// TIA Portal V17 export
// export: Created 2025-04-25T10:07:11.7056769Z, ExportSetting WithDefaults, DisplayName Totally Integrated Automation Portal, DisplayVersion V17 Update 8, DisplayName TIA Portal Openness, DisplayVersion V17 Update 8, DisplayName TIA Portal Version Control Interface, DisplayVersion V17, DisplayName SINAMICS Startdrive Advanced, DisplayVersion V17 SP2, DisplayName SINAMICS Startdrive G110M, G120, G120C, G120D, G120P, G115D, DisplayVersion V17 SP2, DisplayName SINAMICS Startdrive G130, G150, S120, S150, SINAMICS MV, S210, DisplayVersion V17 SP2, DisplayName STEP 7 Professional, DisplayVersion V17 Update 8, DisplayName SINUMERIK ONE STEP 7 Toolbox, DisplayVersion V17 Update 12, DisplayName SINUMERIK 840D sl STEP 7 Toolbox, DisplayVersion V17 Update 12, DisplayName STEP 7 Safety, DisplayVersion V17 Update 6, DisplayName WinCC Advanced / Unified PC, DisplayVersion V17 Update 8
FUNCTION "FC353_NCK_M_CH3_UNIT_1_STA_4" : Void   // FC353, LAD
TITLE = Channel 1 data
{ S7_Optimized_Access := 'FALSE' }
AUTHOR : ETXETAR
VERSION : 1.0
// stored: AutoNumber false, IsIECCheckEnabled false, SetENOAutomatically false, UDAEnableTagReadback false
   VAR_TEMP
      auxm3 : Bool;
      auxm5 : Bool;
   END_VAR
   VAR_TEMP   // added for the SCL form of the ladder/FBD networks
      _w1 : Bool;
      _w2 : Bool;
   END_VAR
BEGIN

REGION Network 1: CALL FB331 M CODE EXTENDED CH4 / M CODE EXTENDED CHANNEL 2
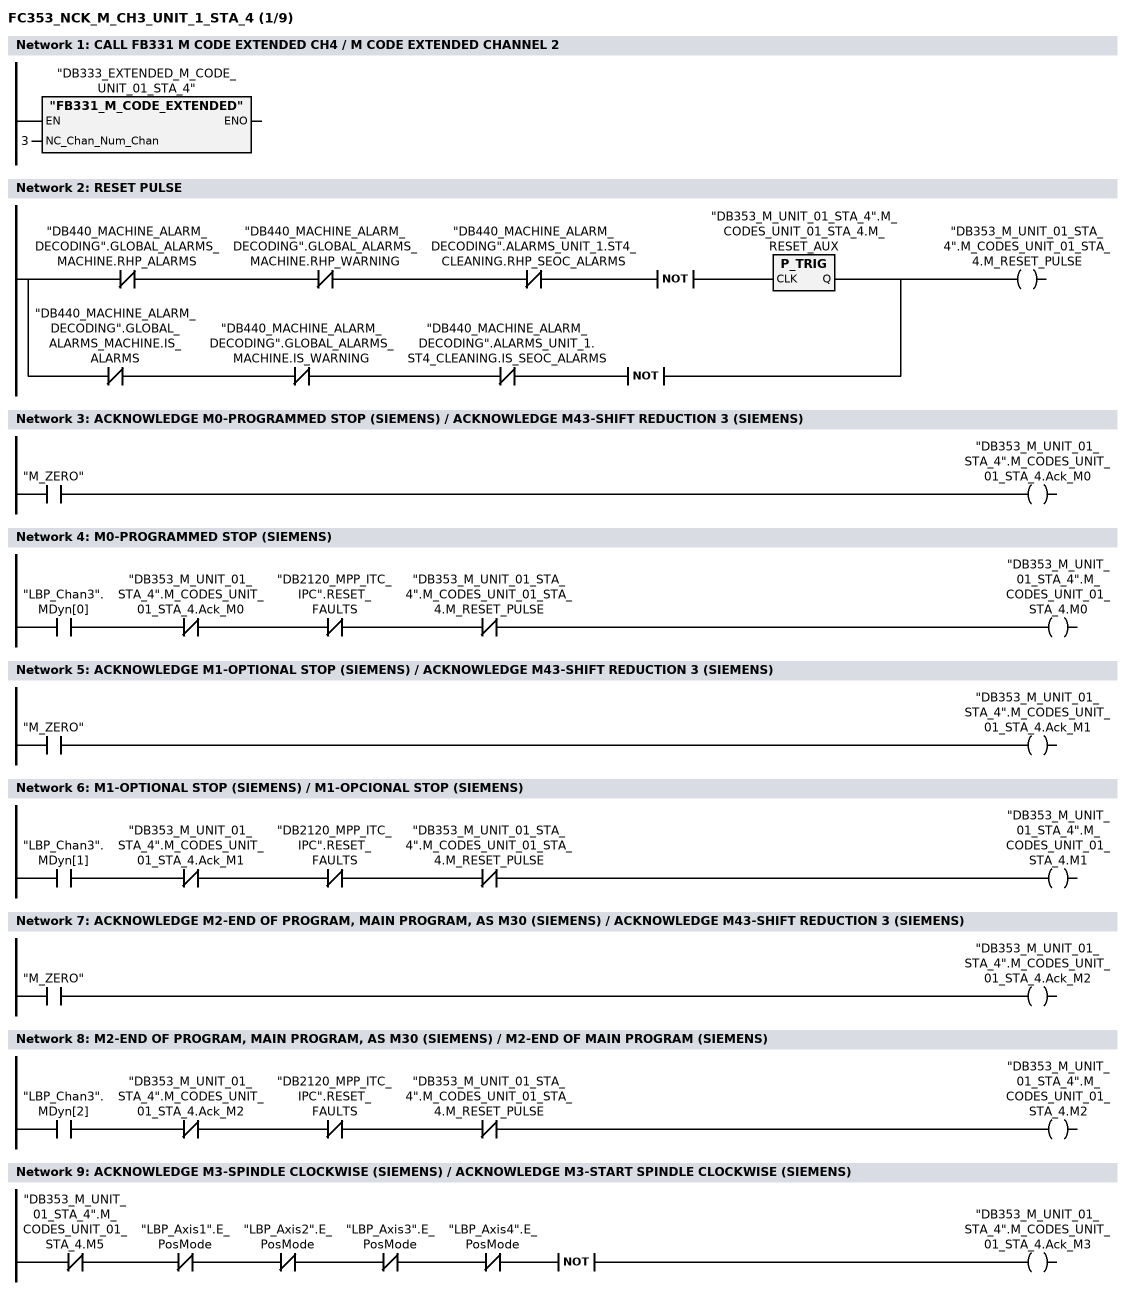
   RUNG wire#powerrail
      "DB333_EXTENDED_M_CODE_UNIT_01_STA_4"(NC_Chan_Num_Chan := 3)
   END_RUNG
   // the same network as SCL:
   "DB333_EXTENDED_M_CODE_UNIT_01_STA_4"(NC_Chan_Num_Chan := 3);   // "FB331_M_CODE_EXTENDED"
END_REGION

REGION Network 2: RESET PULSE
   RUNG wire#powerrail
      I_Contact( "DB440_MACHINE_ALARM_DECODING".GLOBAL_ALARMS_MACHINE.RHP_ALARMS )
      I_Contact( "DB440_MACHINE_ALARM_DECODING".GLOBAL_ALARMS_MACHINE.RHP_WARNING )
      I_Contact( "DB440_MACHINE_ALARM_DECODING".ALARMS_UNIT_1.ST4_CLEANING.RHP_SEOC_ALARMS )
      Not()
      P_Trig( "DB353_M_UNIT_01_STA_4".M_CODES_UNIT_01_STA_4.M_RESET_AUX )
      wire#w1
      Coil( "DB353_M_UNIT_01_STA_4".M_CODES_UNIT_01_STA_4.M_RESET_PULSE )
   END_RUNG
   RUNG wire#powerrail
      I_Contact( "DB440_MACHINE_ALARM_DECODING".GLOBAL_ALARMS_MACHINE.IS_ALARMS )
      I_Contact( "DB440_MACHINE_ALARM_DECODING".GLOBAL_ALARMS_MACHINE.IS_WARNING )
      I_Contact( "DB440_MACHINE_ALARM_DECODING".ALARMS_UNIT_1.ST4_CLEANING.IS_SEOC_ALARMS )
      Not()
   END_RUNG wire#w1
   // the same network as SCL:
   #_w1 := NOT (NOT "DB440_MACHINE_ALARM_DECODING".GLOBAL_ALARMS_MACHINE.RHP_ALARMS AND NOT "DB440_MACHINE_ALARM_DECODING".GLOBAL_ALARMS_MACHINE.RHP_WARNING AND NOT "DB440_MACHINE_ALARM_DECODING".ALARMS_UNIT_1.ST4_CLEANING.RHP_SEOC_ALARMS);
   #_w2 := #_w1 AND NOT "DB353_M_UNIT_01_STA_4".M_CODES_UNIT_01_STA_4.M_RESET_AUX;   // rising edge
   "DB353_M_UNIT_01_STA_4".M_CODES_UNIT_01_STA_4.M_RESET_AUX := #_w1;
   "DB353_M_UNIT_01_STA_4".M_CODES_UNIT_01_STA_4.M_RESET_PULSE := #_w2 OR NOT (NOT "DB440_MACHINE_ALARM_DECODING".GLOBAL_ALARMS_MACHINE.IS_ALARMS AND NOT "DB440_MACHINE_ALARM_DECODING".GLOBAL_ALARMS_MACHINE.IS_WARNING AND NOT "DB440_MACHINE_ALARM_DECODING".ALARMS_UNIT_1.ST4_CLEANING.IS_SEOC_ALARMS);
END_REGION

REGION Network 3: ACKNOWLEDGE M0-PROGRAMMED STOP (SIEMENS) / ACKNOWLEDGE M43-SHIFT REDUCTION 3 (SIEMENS)
   RUNG wire#powerrail
      Contact( "M_ZERO" )
      Coil( "DB353_M_UNIT_01_STA_4".M_CODES_UNIT_01_STA_4.Ack_M0 )
   END_RUNG
   // the same network as SCL:
   "DB353_M_UNIT_01_STA_4".M_CODES_UNIT_01_STA_4.Ack_M0 := "M_ZERO";
END_REGION

REGION Network 4: M0-PROGRAMMED STOP (SIEMENS)
   RUNG wire#powerrail
      Contact( "LBP_Chan3".MDyn[0] )
      I_Contact( "DB353_M_UNIT_01_STA_4".M_CODES_UNIT_01_STA_4.Ack_M0 )
      I_Contact( "DB2120_MPP_ITC_IPC".RESET_FAULTS )
      I_Contact( "DB353_M_UNIT_01_STA_4".M_CODES_UNIT_01_STA_4.M_RESET_PULSE )
      Coil( "DB353_M_UNIT_01_STA_4".M_CODES_UNIT_01_STA_4.M0 )
   END_RUNG
   // the same network as SCL:
   "DB353_M_UNIT_01_STA_4".M_CODES_UNIT_01_STA_4.M0 := "LBP_Chan3".MDyn[0] AND NOT "DB353_M_UNIT_01_STA_4".M_CODES_UNIT_01_STA_4.Ack_M0 AND NOT "DB2120_MPP_ITC_IPC".RESET_FAULTS AND NOT "DB353_M_UNIT_01_STA_4".M_CODES_UNIT_01_STA_4.M_RESET_PULSE;
END_REGION

REGION Network 5: ACKNOWLEDGE M1-OPTIONAL STOP (SIEMENS) / ACKNOWLEDGE M43-SHIFT REDUCTION 3 (SIEMENS)
   RUNG wire#powerrail
      Contact( "M_ZERO" )
      Coil( "DB353_M_UNIT_01_STA_4".M_CODES_UNIT_01_STA_4.Ack_M1 )
   END_RUNG
   // the same network as SCL:
   "DB353_M_UNIT_01_STA_4".M_CODES_UNIT_01_STA_4.Ack_M1 := "M_ZERO";
END_REGION

REGION Network 6: M1-OPTIONAL STOP (SIEMENS) / M1-OPCIONAL STOP (SIEMENS)
   RUNG wire#powerrail
      Contact( "LBP_Chan3".MDyn[1] )
      I_Contact( "DB353_M_UNIT_01_STA_4".M_CODES_UNIT_01_STA_4.Ack_M1 )
      I_Contact( "DB2120_MPP_ITC_IPC".RESET_FAULTS )
      I_Contact( "DB353_M_UNIT_01_STA_4".M_CODES_UNIT_01_STA_4.M_RESET_PULSE )
      Coil( "DB353_M_UNIT_01_STA_4".M_CODES_UNIT_01_STA_4.M1 )
   END_RUNG
   // the same network as SCL:
   "DB353_M_UNIT_01_STA_4".M_CODES_UNIT_01_STA_4.M1 := "LBP_Chan3".MDyn[1] AND NOT "DB353_M_UNIT_01_STA_4".M_CODES_UNIT_01_STA_4.Ack_M1 AND NOT "DB2120_MPP_ITC_IPC".RESET_FAULTS AND NOT "DB353_M_UNIT_01_STA_4".M_CODES_UNIT_01_STA_4.M_RESET_PULSE;
END_REGION

REGION Network 7: ACKNOWLEDGE M2-END OF PROGRAM, MAIN PROGRAM, AS M30 (SIEMENS) / ACKNOWLEDGE M43-SHIFT REDUCTION 3 (SIEMENS)
   RUNG wire#powerrail
      Contact( "M_ZERO" )
      Coil( "DB353_M_UNIT_01_STA_4".M_CODES_UNIT_01_STA_4.Ack_M2 )
   END_RUNG
   // the same network as SCL:
   "DB353_M_UNIT_01_STA_4".M_CODES_UNIT_01_STA_4.Ack_M2 := "M_ZERO";
END_REGION

REGION Network 8: M2-END OF PROGRAM, MAIN PROGRAM, AS M30 (SIEMENS) / M2-END OF MAIN PROGRAM (SIEMENS)
   RUNG wire#powerrail
      Contact( "LBP_Chan3".MDyn[2] )
      I_Contact( "DB353_M_UNIT_01_STA_4".M_CODES_UNIT_01_STA_4.Ack_M2 )
      I_Contact( "DB2120_MPP_ITC_IPC".RESET_FAULTS )
      I_Contact( "DB353_M_UNIT_01_STA_4".M_CODES_UNIT_01_STA_4.M_RESET_PULSE )
      Coil( "DB353_M_UNIT_01_STA_4".M_CODES_UNIT_01_STA_4.M2 )
   END_RUNG
   // the same network as SCL:
   "DB353_M_UNIT_01_STA_4".M_CODES_UNIT_01_STA_4.M2 := "LBP_Chan3".MDyn[2] AND NOT "DB353_M_UNIT_01_STA_4".M_CODES_UNIT_01_STA_4.Ack_M2 AND NOT "DB2120_MPP_ITC_IPC".RESET_FAULTS AND NOT "DB353_M_UNIT_01_STA_4".M_CODES_UNIT_01_STA_4.M_RESET_PULSE;
END_REGION

REGION Network 9: ACKNOWLEDGE M3-SPINDLE CLOCKWISE (SIEMENS) / ACKNOWLEDGE M3-START SPINDLE CLOCKWISE (SIEMENS)
   RUNG wire#powerrail
      I_Contact( "DB353_M_UNIT_01_STA_4".M_CODES_UNIT_01_STA_4.M5 )
      I_Contact( "LBP_Axis1".E_PosMode )
      I_Contact( "LBP_Axis2".E_PosMode )
      I_Contact( "LBP_Axis3".E_PosMode )
      I_Contact( "LBP_Axis4".E_PosMode )
      Not()
      Coil( "DB353_M_UNIT_01_STA_4".M_CODES_UNIT_01_STA_4.Ack_M3 )
   END_RUNG
   // the same network as SCL:
   "DB353_M_UNIT_01_STA_4".M_CODES_UNIT_01_STA_4.Ack_M3 := NOT (NOT "DB353_M_UNIT_01_STA_4".M_CODES_UNIT_01_STA_4.M5 AND NOT "LBP_Axis1".E_PosMode AND NOT "LBP_Axis2".E_PosMode AND NOT "LBP_Axis3".E_PosMode AND NOT "LBP_Axis4".E_PosMode);
END_REGION

REGION Network 10: M3-SPINDLE CLOCKWISE AUXILIARY (SIEMENS) / Extended address M function 1 (16 bit INT)
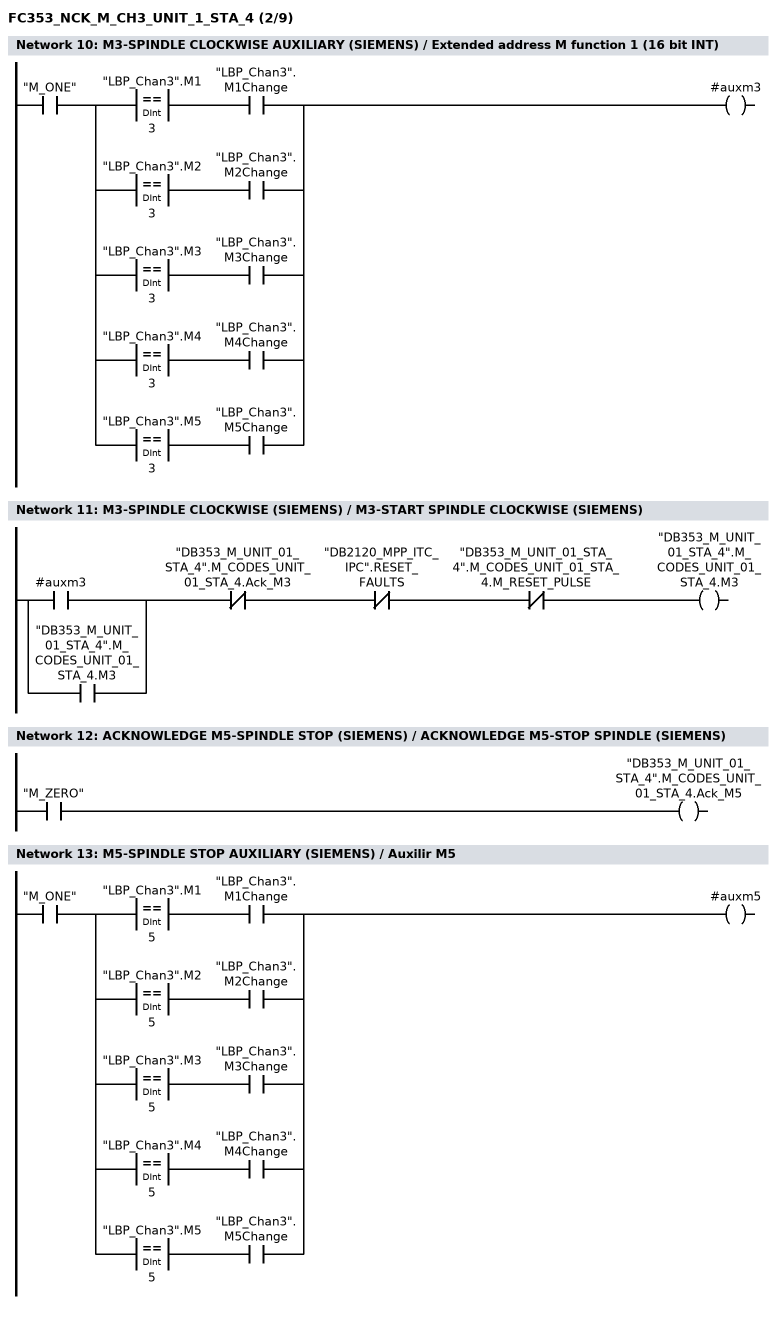
   RUNG wire#powerrail
      Contact( "M_ONE" )
      wire#w1
      { S7_Templates := "SrcType := DInt" } EQ_Contact(in1 := "LBP_Chan3".M1, in2 := 3)
      Contact( "LBP_Chan3".M1Change )
      wire#w2
      Coil( #auxm3 )
   END_RUNG
   RUNG wire#w1
      { S7_Templates := "SrcType := DInt" } EQ_Contact(in1 := "LBP_Chan3".M2, in2 := 3)
      Contact( "LBP_Chan3".M2Change )
   END_RUNG wire#w2
   RUNG wire#w1
      { S7_Templates := "SrcType := DInt" } EQ_Contact(in1 := "LBP_Chan3".M3, in2 := 3)
      Contact( "LBP_Chan3".M3Change )
   END_RUNG wire#w2
   RUNG wire#w1
      { S7_Templates := "SrcType := DInt" } EQ_Contact(in1 := "LBP_Chan3".M4, in2 := 3)
      Contact( "LBP_Chan3".M4Change )
   END_RUNG wire#w2
   RUNG wire#w1
      { S7_Templates := "SrcType := DInt" } EQ_Contact(in1 := "LBP_Chan3".M5, in2 := 3)
      Contact( "LBP_Chan3".M5Change )
   END_RUNG wire#w2
   // the same network as SCL:
   #auxm3 := "M_ONE" AND ((("LBP_Chan3".M1 = 3) AND "LBP_Chan3".M1Change) OR (("LBP_Chan3".M2 = 3) AND "LBP_Chan3".M2Change) OR (("LBP_Chan3".M3 = 3) AND "LBP_Chan3".M3Change) OR (("LBP_Chan3".M4 = 3) AND "LBP_Chan3".M4Change) OR (("LBP_Chan3".M5 = 3) AND "LBP_Chan3".M5Change));
END_REGION

REGION Network 11: M3-SPINDLE CLOCKWISE (SIEMENS) / M3-START SPINDLE CLOCKWISE (SIEMENS)
   RUNG wire#powerrail
      Contact( #auxm3 )
      wire#w1
      I_Contact( "DB353_M_UNIT_01_STA_4".M_CODES_UNIT_01_STA_4.Ack_M3 )
      I_Contact( "DB2120_MPP_ITC_IPC".RESET_FAULTS )
      I_Contact( "DB353_M_UNIT_01_STA_4".M_CODES_UNIT_01_STA_4.M_RESET_PULSE )
      Coil( "DB353_M_UNIT_01_STA_4".M_CODES_UNIT_01_STA_4.M3 )
   END_RUNG
   RUNG wire#powerrail
      Contact( "DB353_M_UNIT_01_STA_4".M_CODES_UNIT_01_STA_4.M3 )
   END_RUNG wire#w1
   // the same network as SCL:
   "DB353_M_UNIT_01_STA_4".M_CODES_UNIT_01_STA_4.M3 := (#auxm3 OR "DB353_M_UNIT_01_STA_4".M_CODES_UNIT_01_STA_4.M3) AND NOT "DB353_M_UNIT_01_STA_4".M_CODES_UNIT_01_STA_4.Ack_M3 AND NOT "DB2120_MPP_ITC_IPC".RESET_FAULTS AND NOT "DB353_M_UNIT_01_STA_4".M_CODES_UNIT_01_STA_4.M_RESET_PULSE;
END_REGION

REGION Network 12: ACKNOWLEDGE M5-SPINDLE STOP (SIEMENS) / ACKNOWLEDGE M5-STOP SPINDLE (SIEMENS)
   RUNG wire#powerrail
      Contact( "M_ZERO" )
      Coil( "DB353_M_UNIT_01_STA_4".M_CODES_UNIT_01_STA_4.Ack_M5 )
   END_RUNG
   // the same network as SCL:
   "DB353_M_UNIT_01_STA_4".M_CODES_UNIT_01_STA_4.Ack_M5 := "M_ZERO";
END_REGION

REGION Network 13: M5-SPINDLE STOP AUXILIARY (SIEMENS) / Auxilir M5
   RUNG wire#powerrail
      Contact( "M_ONE" )
      wire#w1
      { S7_Templates := "SrcType := DInt" } EQ_Contact(in1 := "LBP_Chan3".M1, in2 := 5)
      Contact( "LBP_Chan3".M1Change )
      wire#w2
      Coil( #auxm5 )
   END_RUNG
   RUNG wire#w1
      { S7_Templates := "SrcType := DInt" } EQ_Contact(in1 := "LBP_Chan3".M2, in2 := 5)
      Contact( "LBP_Chan3".M2Change )
   END_RUNG wire#w2
   RUNG wire#w1
      { S7_Templates := "SrcType := DInt" } EQ_Contact(in1 := "LBP_Chan3".M3, in2 := 5)
      Contact( "LBP_Chan3".M3Change )
   END_RUNG wire#w2
   RUNG wire#w1
      { S7_Templates := "SrcType := DInt" } EQ_Contact(in1 := "LBP_Chan3".M4, in2 := 5)
      Contact( "LBP_Chan3".M4Change )
   END_RUNG wire#w2
   RUNG wire#w1
      { S7_Templates := "SrcType := DInt" } EQ_Contact(in1 := "LBP_Chan3".M5, in2 := 5)
      Contact( "LBP_Chan3".M5Change )
   END_RUNG wire#w2
   // the same network as SCL:
   #auxm5 := "M_ONE" AND ((("LBP_Chan3".M1 = 5) AND "LBP_Chan3".M1Change) OR (("LBP_Chan3".M2 = 5) AND "LBP_Chan3".M2Change) OR (("LBP_Chan3".M3 = 5) AND "LBP_Chan3".M3Change) OR (("LBP_Chan3".M4 = 5) AND "LBP_Chan3".M4Change) OR (("LBP_Chan3".M5 = 5) AND "LBP_Chan3".M5Change));
END_REGION

REGION Network 14: M5-SPINDLE STOP (SIEMENS) / M5-STOP SPINDLE (SIEMENS)
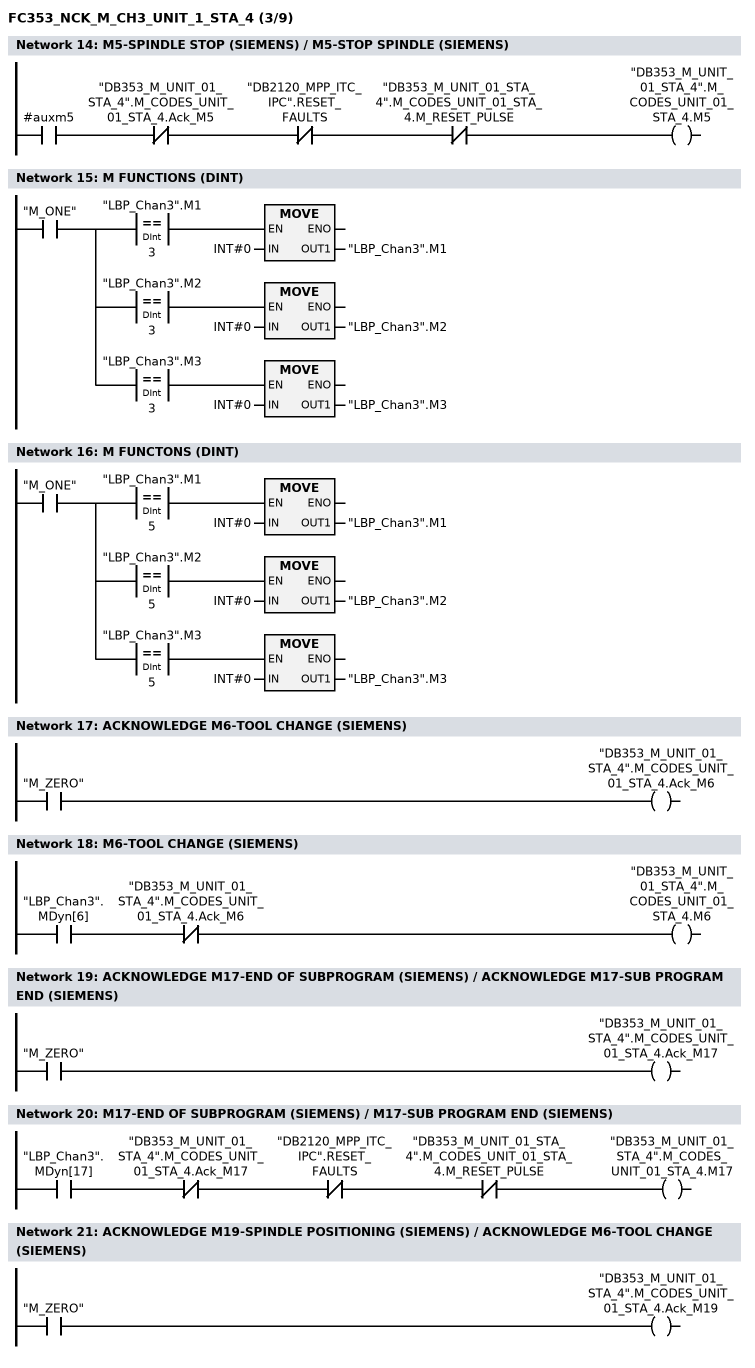
   RUNG wire#powerrail
      Contact( #auxm5 )
      I_Contact( "DB353_M_UNIT_01_STA_4".M_CODES_UNIT_01_STA_4.Ack_M5 )
      I_Contact( "DB2120_MPP_ITC_IPC".RESET_FAULTS )
      I_Contact( "DB353_M_UNIT_01_STA_4".M_CODES_UNIT_01_STA_4.M_RESET_PULSE )
      Coil( "DB353_M_UNIT_01_STA_4".M_CODES_UNIT_01_STA_4.M5 )
   END_RUNG
   // the same network as SCL:
   "DB353_M_UNIT_01_STA_4".M_CODES_UNIT_01_STA_4.M5 := #auxm5 AND NOT "DB353_M_UNIT_01_STA_4".M_CODES_UNIT_01_STA_4.Ack_M5 AND NOT "DB2120_MPP_ITC_IPC".RESET_FAULTS AND NOT "DB353_M_UNIT_01_STA_4".M_CODES_UNIT_01_STA_4.M_RESET_PULSE;
END_REGION

REGION Network 15: M FUNCTIONS (DINT)
   RUNG wire#powerrail
      Contact( "M_ONE" )
      wire#w1
      { S7_Templates := "SrcType := DInt" } EQ_Contact(in1 := "LBP_Chan3".M1, in2 := 3)
      { S7_GenerateENO := "TRUE" } Move(in := INT#0, out1 => "LBP_Chan3".M1)
   END_RUNG
   RUNG wire#w1
      { S7_Templates := "SrcType := DInt" } EQ_Contact(in1 := "LBP_Chan3".M2, in2 := 3)
      { S7_GenerateENO := "TRUE" } Move(in := INT#0, out1 => "LBP_Chan3".M2)
   END_RUNG
   RUNG wire#w1
      { S7_Templates := "SrcType := DInt" } EQ_Contact(in1 := "LBP_Chan3".M3, in2 := 3)
      { S7_GenerateENO := "TRUE" } Move(in := INT#0, out1 => "LBP_Chan3".M3)
   END_RUNG
   // the same network as SCL:
   IF "M_ONE" AND ("LBP_Chan3".M1 = 3) THEN "LBP_Chan3".M1 := INT#0; END_IF;
   IF "M_ONE" AND ("LBP_Chan3".M2 = 3) THEN "LBP_Chan3".M2 := INT#0; END_IF;
   IF "M_ONE" AND ("LBP_Chan3".M3 = 3) THEN "LBP_Chan3".M3 := INT#0; END_IF;
END_REGION

REGION Network 16: M FUNCTONS (DINT)
   RUNG wire#powerrail
      Contact( "M_ONE" )
      wire#w1
      { S7_Templates := "SrcType := DInt" } EQ_Contact(in1 := "LBP_Chan3".M1, in2 := 5)
      { S7_GenerateENO := "TRUE" } Move(in := INT#0, out1 => "LBP_Chan3".M1)
   END_RUNG
   RUNG wire#w1
      { S7_Templates := "SrcType := DInt" } EQ_Contact(in1 := "LBP_Chan3".M2, in2 := 5)
      { S7_GenerateENO := "TRUE" } Move(in := INT#0, out1 => "LBP_Chan3".M2)
   END_RUNG
   RUNG wire#w1
      { S7_Templates := "SrcType := DInt" } EQ_Contact(in1 := "LBP_Chan3".M3, in2 := 5)
      { S7_GenerateENO := "TRUE" } Move(in := INT#0, out1 => "LBP_Chan3".M3)
   END_RUNG
   // the same network as SCL:
   IF "M_ONE" AND ("LBP_Chan3".M1 = 5) THEN "LBP_Chan3".M1 := INT#0; END_IF;
   IF "M_ONE" AND ("LBP_Chan3".M2 = 5) THEN "LBP_Chan3".M2 := INT#0; END_IF;
   IF "M_ONE" AND ("LBP_Chan3".M3 = 5) THEN "LBP_Chan3".M3 := INT#0; END_IF;
END_REGION

REGION Network 17: ACKNOWLEDGE M6-TOOL CHANGE (SIEMENS)
   RUNG wire#powerrail
      Contact( "M_ZERO" )
      Coil( "DB353_M_UNIT_01_STA_4".M_CODES_UNIT_01_STA_4.Ack_M6 )
   END_RUNG
   // the same network as SCL:
   "DB353_M_UNIT_01_STA_4".M_CODES_UNIT_01_STA_4.Ack_M6 := "M_ZERO";
END_REGION

REGION Network 18: M6-TOOL CHANGE (SIEMENS)
   RUNG wire#powerrail
      Contact( "LBP_Chan3".MDyn[6] )
      I_Contact( "DB353_M_UNIT_01_STA_4".M_CODES_UNIT_01_STA_4.Ack_M6 )
      Coil( "DB353_M_UNIT_01_STA_4".M_CODES_UNIT_01_STA_4.M6 )
   END_RUNG
   // the same network as SCL:
   "DB353_M_UNIT_01_STA_4".M_CODES_UNIT_01_STA_4.M6 := "LBP_Chan3".MDyn[6] AND NOT "DB353_M_UNIT_01_STA_4".M_CODES_UNIT_01_STA_4.Ack_M6;
END_REGION

REGION Network 19: ACKNOWLEDGE M17-END OF SUBPROGRAM (SIEMENS) / ACKNOWLEDGE M17-SUB PROGRAM END (SIEMENS)
   RUNG wire#powerrail
      Contact( "M_ZERO" )
      Coil( "DB353_M_UNIT_01_STA_4".M_CODES_UNIT_01_STA_4.Ack_M17 )
   END_RUNG
   // the same network as SCL:
   "DB353_M_UNIT_01_STA_4".M_CODES_UNIT_01_STA_4.Ack_M17 := "M_ZERO";
END_REGION

REGION Network 20: M17-END OF SUBPROGRAM (SIEMENS) / M17-SUB PROGRAM END (SIEMENS)
   RUNG wire#powerrail
      Contact( "LBP_Chan3".MDyn[17] )
      I_Contact( "DB353_M_UNIT_01_STA_4".M_CODES_UNIT_01_STA_4.Ack_M17 )
      I_Contact( "DB2120_MPP_ITC_IPC".RESET_FAULTS )
      I_Contact( "DB353_M_UNIT_01_STA_4".M_CODES_UNIT_01_STA_4.M_RESET_PULSE )
      Coil( "DB353_M_UNIT_01_STA_4".M_CODES_UNIT_01_STA_4.M17 )
   END_RUNG
   // the same network as SCL:
   "DB353_M_UNIT_01_STA_4".M_CODES_UNIT_01_STA_4.M17 := "LBP_Chan3".MDyn[17] AND NOT "DB353_M_UNIT_01_STA_4".M_CODES_UNIT_01_STA_4.Ack_M17 AND NOT "DB2120_MPP_ITC_IPC".RESET_FAULTS AND NOT "DB353_M_UNIT_01_STA_4".M_CODES_UNIT_01_STA_4.M_RESET_PULSE;
END_REGION

REGION Network 21: ACKNOWLEDGE M19-SPINDLE POSITIONING (SIEMENS) / ACKNOWLEDGE M6-TOOL CHANGE (SIEMENS)
   RUNG wire#powerrail
      Contact( "M_ZERO" )
      Coil( "DB353_M_UNIT_01_STA_4".M_CODES_UNIT_01_STA_4.Ack_M19 )
   END_RUNG
   // the same network as SCL:
   "DB353_M_UNIT_01_STA_4".M_CODES_UNIT_01_STA_4.Ack_M19 := "M_ZERO";
END_REGION

REGION Network 22: M19-SPINDLE POSITIONING (SIEMENS) / M6-TOOL CHANGE (SIEMENS)
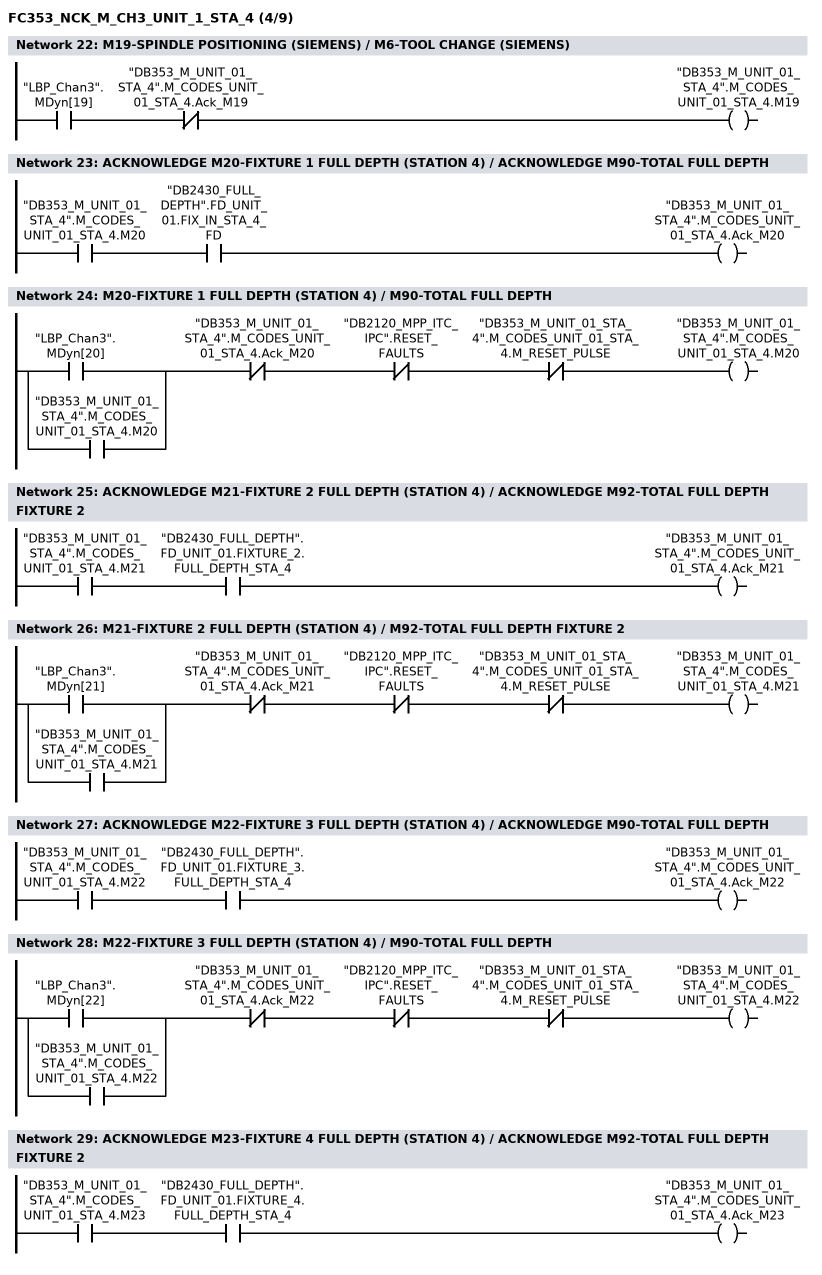
   RUNG wire#powerrail
      Contact( "LBP_Chan3".MDyn[19] )
      I_Contact( "DB353_M_UNIT_01_STA_4".M_CODES_UNIT_01_STA_4.Ack_M19 )
      Coil( "DB353_M_UNIT_01_STA_4".M_CODES_UNIT_01_STA_4.M19 )
   END_RUNG
   // the same network as SCL:
   "DB353_M_UNIT_01_STA_4".M_CODES_UNIT_01_STA_4.M19 := "LBP_Chan3".MDyn[19] AND NOT "DB353_M_UNIT_01_STA_4".M_CODES_UNIT_01_STA_4.Ack_M19;
END_REGION

REGION Network 23: ACKNOWLEDGE M20-FIXTURE 1 FULL DEPTH (STATION 4) / ACKNOWLEDGE M90-TOTAL FULL DEPTH
   RUNG wire#powerrail
      Contact( "DB353_M_UNIT_01_STA_4".M_CODES_UNIT_01_STA_4.M20 )
      Contact( "DB2430_FULL_DEPTH".FD_UNIT_01.FIX_IN_STA_4_FD )
      Coil( "DB353_M_UNIT_01_STA_4".M_CODES_UNIT_01_STA_4.Ack_M20 )
   END_RUNG
   // the same network as SCL:
   "DB353_M_UNIT_01_STA_4".M_CODES_UNIT_01_STA_4.Ack_M20 := "DB353_M_UNIT_01_STA_4".M_CODES_UNIT_01_STA_4.M20 AND "DB2430_FULL_DEPTH".FD_UNIT_01.FIX_IN_STA_4_FD;
END_REGION

REGION Network 24: M20-FIXTURE 1 FULL DEPTH (STATION 4) / M90-TOTAL FULL DEPTH
   RUNG wire#powerrail
      Contact( "LBP_Chan3".MDyn[20] )
      wire#w1
      I_Contact( "DB353_M_UNIT_01_STA_4".M_CODES_UNIT_01_STA_4.Ack_M20 )
      I_Contact( "DB2120_MPP_ITC_IPC".RESET_FAULTS )
      I_Contact( "DB353_M_UNIT_01_STA_4".M_CODES_UNIT_01_STA_4.M_RESET_PULSE )
      Coil( "DB353_M_UNIT_01_STA_4".M_CODES_UNIT_01_STA_4.M20 )
   END_RUNG
   RUNG wire#powerrail
      Contact( "DB353_M_UNIT_01_STA_4".M_CODES_UNIT_01_STA_4.M20 )
   END_RUNG wire#w1
   // the same network as SCL:
   "DB353_M_UNIT_01_STA_4".M_CODES_UNIT_01_STA_4.M20 := ("LBP_Chan3".MDyn[20] OR "DB353_M_UNIT_01_STA_4".M_CODES_UNIT_01_STA_4.M20) AND NOT "DB353_M_UNIT_01_STA_4".M_CODES_UNIT_01_STA_4.Ack_M20 AND NOT "DB2120_MPP_ITC_IPC".RESET_FAULTS AND NOT "DB353_M_UNIT_01_STA_4".M_CODES_UNIT_01_STA_4.M_RESET_PULSE;
END_REGION

REGION Network 25: ACKNOWLEDGE M21-FIXTURE 2 FULL DEPTH (STATION 4) / ACKNOWLEDGE M92-TOTAL FULL DEPTH FIXTURE 2
   RUNG wire#powerrail
      Contact( "DB353_M_UNIT_01_STA_4".M_CODES_UNIT_01_STA_4.M21 )
      Contact( "DB2430_FULL_DEPTH".FD_UNIT_01.FIXTURE_2.FULL_DEPTH_STA_4 )
      Coil( "DB353_M_UNIT_01_STA_4".M_CODES_UNIT_01_STA_4.Ack_M21 )
   END_RUNG
   // the same network as SCL:
   "DB353_M_UNIT_01_STA_4".M_CODES_UNIT_01_STA_4.Ack_M21 := "DB353_M_UNIT_01_STA_4".M_CODES_UNIT_01_STA_4.M21 AND "DB2430_FULL_DEPTH".FD_UNIT_01.FIXTURE_2.FULL_DEPTH_STA_4;
END_REGION

REGION Network 26: M21-FIXTURE 2 FULL DEPTH (STATION 4) / M92-TOTAL FULL DEPTH FIXTURE 2
   RUNG wire#powerrail
      Contact( "LBP_Chan3".MDyn[21] )
      wire#w1
      I_Contact( "DB353_M_UNIT_01_STA_4".M_CODES_UNIT_01_STA_4.Ack_M21 )
      I_Contact( "DB2120_MPP_ITC_IPC".RESET_FAULTS )
      I_Contact( "DB353_M_UNIT_01_STA_4".M_CODES_UNIT_01_STA_4.M_RESET_PULSE )
      Coil( "DB353_M_UNIT_01_STA_4".M_CODES_UNIT_01_STA_4.M21 )
   END_RUNG
   RUNG wire#powerrail
      Contact( "DB353_M_UNIT_01_STA_4".M_CODES_UNIT_01_STA_4.M21 )
   END_RUNG wire#w1
   // the same network as SCL:
   "DB353_M_UNIT_01_STA_4".M_CODES_UNIT_01_STA_4.M21 := ("LBP_Chan3".MDyn[21] OR "DB353_M_UNIT_01_STA_4".M_CODES_UNIT_01_STA_4.M21) AND NOT "DB353_M_UNIT_01_STA_4".M_CODES_UNIT_01_STA_4.Ack_M21 AND NOT "DB2120_MPP_ITC_IPC".RESET_FAULTS AND NOT "DB353_M_UNIT_01_STA_4".M_CODES_UNIT_01_STA_4.M_RESET_PULSE;
END_REGION

REGION Network 27: ACKNOWLEDGE M22-FIXTURE 3 FULL DEPTH (STATION 4) / ACKNOWLEDGE M90-TOTAL FULL DEPTH
   RUNG wire#powerrail
      Contact( "DB353_M_UNIT_01_STA_4".M_CODES_UNIT_01_STA_4.M22 )
      Contact( "DB2430_FULL_DEPTH".FD_UNIT_01.FIXTURE_3.FULL_DEPTH_STA_4 )
      Coil( "DB353_M_UNIT_01_STA_4".M_CODES_UNIT_01_STA_4.Ack_M22 )
   END_RUNG
   // the same network as SCL:
   "DB353_M_UNIT_01_STA_4".M_CODES_UNIT_01_STA_4.Ack_M22 := "DB353_M_UNIT_01_STA_4".M_CODES_UNIT_01_STA_4.M22 AND "DB2430_FULL_DEPTH".FD_UNIT_01.FIXTURE_3.FULL_DEPTH_STA_4;
END_REGION

REGION Network 28: M22-FIXTURE 3 FULL DEPTH (STATION 4) / M90-TOTAL FULL DEPTH
   RUNG wire#powerrail
      Contact( "LBP_Chan3".MDyn[22] )
      wire#w1
      I_Contact( "DB353_M_UNIT_01_STA_4".M_CODES_UNIT_01_STA_4.Ack_M22 )
      I_Contact( "DB2120_MPP_ITC_IPC".RESET_FAULTS )
      I_Contact( "DB353_M_UNIT_01_STA_4".M_CODES_UNIT_01_STA_4.M_RESET_PULSE )
      Coil( "DB353_M_UNIT_01_STA_4".M_CODES_UNIT_01_STA_4.M22 )
   END_RUNG
   RUNG wire#powerrail
      Contact( "DB353_M_UNIT_01_STA_4".M_CODES_UNIT_01_STA_4.M22 )
   END_RUNG wire#w1
   // the same network as SCL:
   "DB353_M_UNIT_01_STA_4".M_CODES_UNIT_01_STA_4.M22 := ("LBP_Chan3".MDyn[22] OR "DB353_M_UNIT_01_STA_4".M_CODES_UNIT_01_STA_4.M22) AND NOT "DB353_M_UNIT_01_STA_4".M_CODES_UNIT_01_STA_4.Ack_M22 AND NOT "DB2120_MPP_ITC_IPC".RESET_FAULTS AND NOT "DB353_M_UNIT_01_STA_4".M_CODES_UNIT_01_STA_4.M_RESET_PULSE;
END_REGION

REGION Network 29: ACKNOWLEDGE M23-FIXTURE 4 FULL DEPTH (STATION 4) / ACKNOWLEDGE M92-TOTAL FULL DEPTH FIXTURE 2
   RUNG wire#powerrail
      Contact( "DB353_M_UNIT_01_STA_4".M_CODES_UNIT_01_STA_4.M23 )
      Contact( "DB2430_FULL_DEPTH".FD_UNIT_01.FIXTURE_4.FULL_DEPTH_STA_4 )
      Coil( "DB353_M_UNIT_01_STA_4".M_CODES_UNIT_01_STA_4.Ack_M23 )
   END_RUNG
   // the same network as SCL:
   "DB353_M_UNIT_01_STA_4".M_CODES_UNIT_01_STA_4.Ack_M23 := "DB353_M_UNIT_01_STA_4".M_CODES_UNIT_01_STA_4.M23 AND "DB2430_FULL_DEPTH".FD_UNIT_01.FIXTURE_4.FULL_DEPTH_STA_4;
END_REGION

REGION Network 30: M23-FIXTURE 4 FULL DEPTH (STATION 4) / M92-TOTAL FULL DEPTH FIXTURE 2
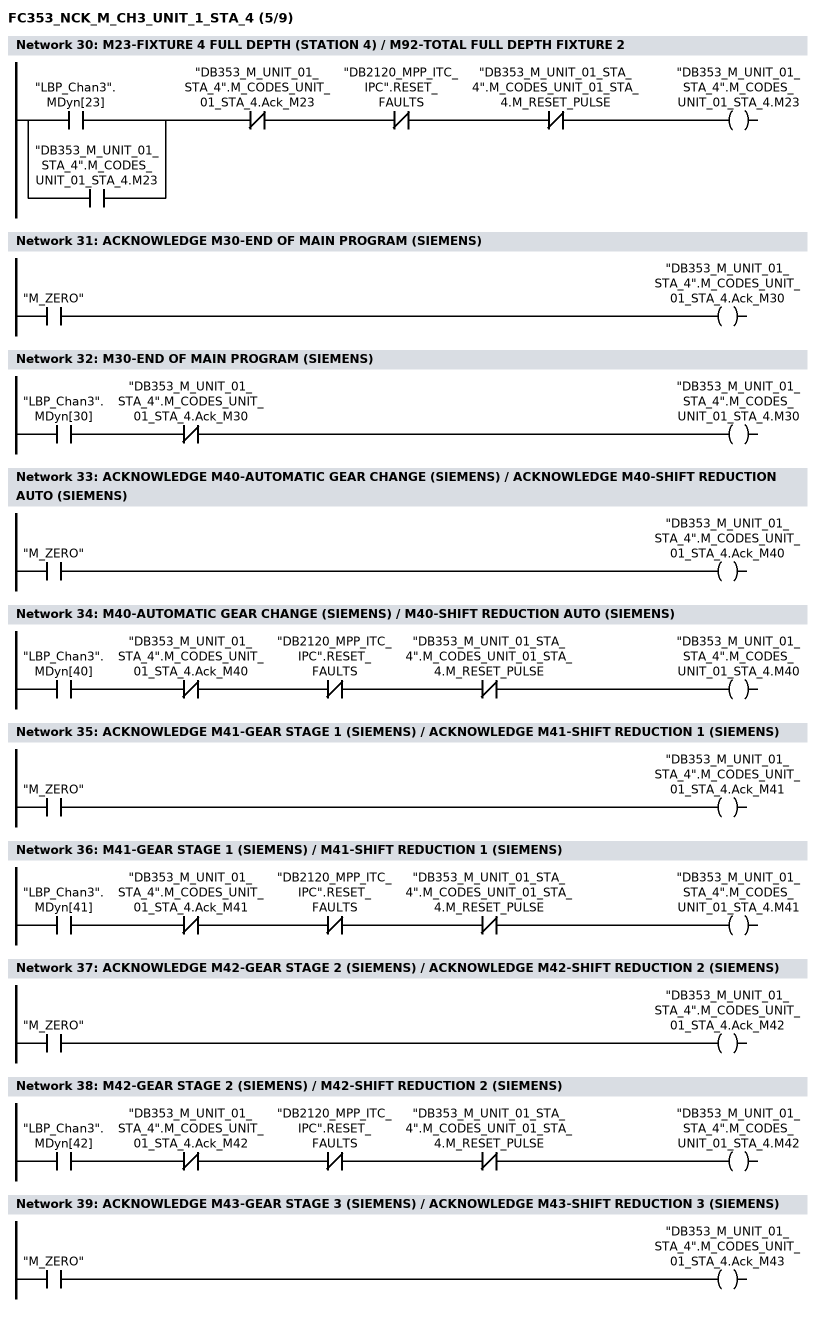
   RUNG wire#powerrail
      Contact( "LBP_Chan3".MDyn[23] )
      wire#w1
      I_Contact( "DB353_M_UNIT_01_STA_4".M_CODES_UNIT_01_STA_4.Ack_M23 )
      I_Contact( "DB2120_MPP_ITC_IPC".RESET_FAULTS )
      I_Contact( "DB353_M_UNIT_01_STA_4".M_CODES_UNIT_01_STA_4.M_RESET_PULSE )
      Coil( "DB353_M_UNIT_01_STA_4".M_CODES_UNIT_01_STA_4.M23 )
   END_RUNG
   RUNG wire#powerrail
      Contact( "DB353_M_UNIT_01_STA_4".M_CODES_UNIT_01_STA_4.M23 )
   END_RUNG wire#w1
   // the same network as SCL:
   "DB353_M_UNIT_01_STA_4".M_CODES_UNIT_01_STA_4.M23 := ("LBP_Chan3".MDyn[23] OR "DB353_M_UNIT_01_STA_4".M_CODES_UNIT_01_STA_4.M23) AND NOT "DB353_M_UNIT_01_STA_4".M_CODES_UNIT_01_STA_4.Ack_M23 AND NOT "DB2120_MPP_ITC_IPC".RESET_FAULTS AND NOT "DB353_M_UNIT_01_STA_4".M_CODES_UNIT_01_STA_4.M_RESET_PULSE;
END_REGION

REGION Network 31: ACKNOWLEDGE M30-END OF MAIN PROGRAM (SIEMENS)
   RUNG wire#powerrail
      Contact( "M_ZERO" )
      Coil( "DB353_M_UNIT_01_STA_4".M_CODES_UNIT_01_STA_4.Ack_M30 )
   END_RUNG
   // the same network as SCL:
   "DB353_M_UNIT_01_STA_4".M_CODES_UNIT_01_STA_4.Ack_M30 := "M_ZERO";
END_REGION

REGION Network 32: M30-END OF MAIN PROGRAM (SIEMENS)
   RUNG wire#powerrail
      Contact( "LBP_Chan3".MDyn[30] )
      I_Contact( "DB353_M_UNIT_01_STA_4".M_CODES_UNIT_01_STA_4.Ack_M30 )
      Coil( "DB353_M_UNIT_01_STA_4".M_CODES_UNIT_01_STA_4.M30 )
   END_RUNG
   // the same network as SCL:
   "DB353_M_UNIT_01_STA_4".M_CODES_UNIT_01_STA_4.M30 := "LBP_Chan3".MDyn[30] AND NOT "DB353_M_UNIT_01_STA_4".M_CODES_UNIT_01_STA_4.Ack_M30;
END_REGION

REGION Network 33: ACKNOWLEDGE M40-AUTOMATIC GEAR CHANGE (SIEMENS) / ACKNOWLEDGE M40-SHIFT REDUCTION AUTO (SIEMENS)
   RUNG wire#powerrail
      Contact( "M_ZERO" )
      Coil( "DB353_M_UNIT_01_STA_4".M_CODES_UNIT_01_STA_4.Ack_M40 )
   END_RUNG
   // the same network as SCL:
   "DB353_M_UNIT_01_STA_4".M_CODES_UNIT_01_STA_4.Ack_M40 := "M_ZERO";
END_REGION

REGION Network 34: M40-AUTOMATIC GEAR CHANGE (SIEMENS) / M40-SHIFT REDUCTION AUTO (SIEMENS)
   RUNG wire#powerrail
      Contact( "LBP_Chan3".MDyn[40] )
      I_Contact( "DB353_M_UNIT_01_STA_4".M_CODES_UNIT_01_STA_4.Ack_M40 )
      I_Contact( "DB2120_MPP_ITC_IPC".RESET_FAULTS )
      I_Contact( "DB353_M_UNIT_01_STA_4".M_CODES_UNIT_01_STA_4.M_RESET_PULSE )
      Coil( "DB353_M_UNIT_01_STA_4".M_CODES_UNIT_01_STA_4.M40 )
   END_RUNG
   // the same network as SCL:
   "DB353_M_UNIT_01_STA_4".M_CODES_UNIT_01_STA_4.M40 := "LBP_Chan3".MDyn[40] AND NOT "DB353_M_UNIT_01_STA_4".M_CODES_UNIT_01_STA_4.Ack_M40 AND NOT "DB2120_MPP_ITC_IPC".RESET_FAULTS AND NOT "DB353_M_UNIT_01_STA_4".M_CODES_UNIT_01_STA_4.M_RESET_PULSE;
END_REGION

REGION Network 35: ACKNOWLEDGE M41-GEAR STAGE 1 (SIEMENS) / ACKNOWLEDGE M41-SHIFT REDUCTION 1 (SIEMENS)
   RUNG wire#powerrail
      Contact( "M_ZERO" )
      Coil( "DB353_M_UNIT_01_STA_4".M_CODES_UNIT_01_STA_4.Ack_M41 )
   END_RUNG
   // the same network as SCL:
   "DB353_M_UNIT_01_STA_4".M_CODES_UNIT_01_STA_4.Ack_M41 := "M_ZERO";
END_REGION

REGION Network 36: M41-GEAR STAGE 1 (SIEMENS) / M41-SHIFT REDUCTION 1 (SIEMENS)
   RUNG wire#powerrail
      Contact( "LBP_Chan3".MDyn[41] )
      I_Contact( "DB353_M_UNIT_01_STA_4".M_CODES_UNIT_01_STA_4.Ack_M41 )
      I_Contact( "DB2120_MPP_ITC_IPC".RESET_FAULTS )
      I_Contact( "DB353_M_UNIT_01_STA_4".M_CODES_UNIT_01_STA_4.M_RESET_PULSE )
      Coil( "DB353_M_UNIT_01_STA_4".M_CODES_UNIT_01_STA_4.M41 )
   END_RUNG
   // the same network as SCL:
   "DB353_M_UNIT_01_STA_4".M_CODES_UNIT_01_STA_4.M41 := "LBP_Chan3".MDyn[41] AND NOT "DB353_M_UNIT_01_STA_4".M_CODES_UNIT_01_STA_4.Ack_M41 AND NOT "DB2120_MPP_ITC_IPC".RESET_FAULTS AND NOT "DB353_M_UNIT_01_STA_4".M_CODES_UNIT_01_STA_4.M_RESET_PULSE;
END_REGION

REGION Network 37: ACKNOWLEDGE M42-GEAR STAGE 2 (SIEMENS) / ACKNOWLEDGE M42-SHIFT REDUCTION 2 (SIEMENS)
   RUNG wire#powerrail
      Contact( "M_ZERO" )
      Coil( "DB353_M_UNIT_01_STA_4".M_CODES_UNIT_01_STA_4.Ack_M42 )
   END_RUNG
   // the same network as SCL:
   "DB353_M_UNIT_01_STA_4".M_CODES_UNIT_01_STA_4.Ack_M42 := "M_ZERO";
END_REGION

REGION Network 38: M42-GEAR STAGE 2 (SIEMENS) / M42-SHIFT REDUCTION 2 (SIEMENS)
   RUNG wire#powerrail
      Contact( "LBP_Chan3".MDyn[42] )
      I_Contact( "DB353_M_UNIT_01_STA_4".M_CODES_UNIT_01_STA_4.Ack_M42 )
      I_Contact( "DB2120_MPP_ITC_IPC".RESET_FAULTS )
      I_Contact( "DB353_M_UNIT_01_STA_4".M_CODES_UNIT_01_STA_4.M_RESET_PULSE )
      Coil( "DB353_M_UNIT_01_STA_4".M_CODES_UNIT_01_STA_4.M42 )
   END_RUNG
   // the same network as SCL:
   "DB353_M_UNIT_01_STA_4".M_CODES_UNIT_01_STA_4.M42 := "LBP_Chan3".MDyn[42] AND NOT "DB353_M_UNIT_01_STA_4".M_CODES_UNIT_01_STA_4.Ack_M42 AND NOT "DB2120_MPP_ITC_IPC".RESET_FAULTS AND NOT "DB353_M_UNIT_01_STA_4".M_CODES_UNIT_01_STA_4.M_RESET_PULSE;
END_REGION

REGION Network 39: ACKNOWLEDGE M43-GEAR STAGE 3 (SIEMENS) / ACKNOWLEDGE M43-SHIFT REDUCTION 3 (SIEMENS)
   RUNG wire#powerrail
      Contact( "M_ZERO" )
      Coil( "DB353_M_UNIT_01_STA_4".M_CODES_UNIT_01_STA_4.Ack_M43 )
   END_RUNG
   // the same network as SCL:
   "DB353_M_UNIT_01_STA_4".M_CODES_UNIT_01_STA_4.Ack_M43 := "M_ZERO";
END_REGION

REGION Network 40: M43-GEAR STAGE 3 (SIEMENS) / M43-SHIFT REDUCTION 3 (SIEMENS)
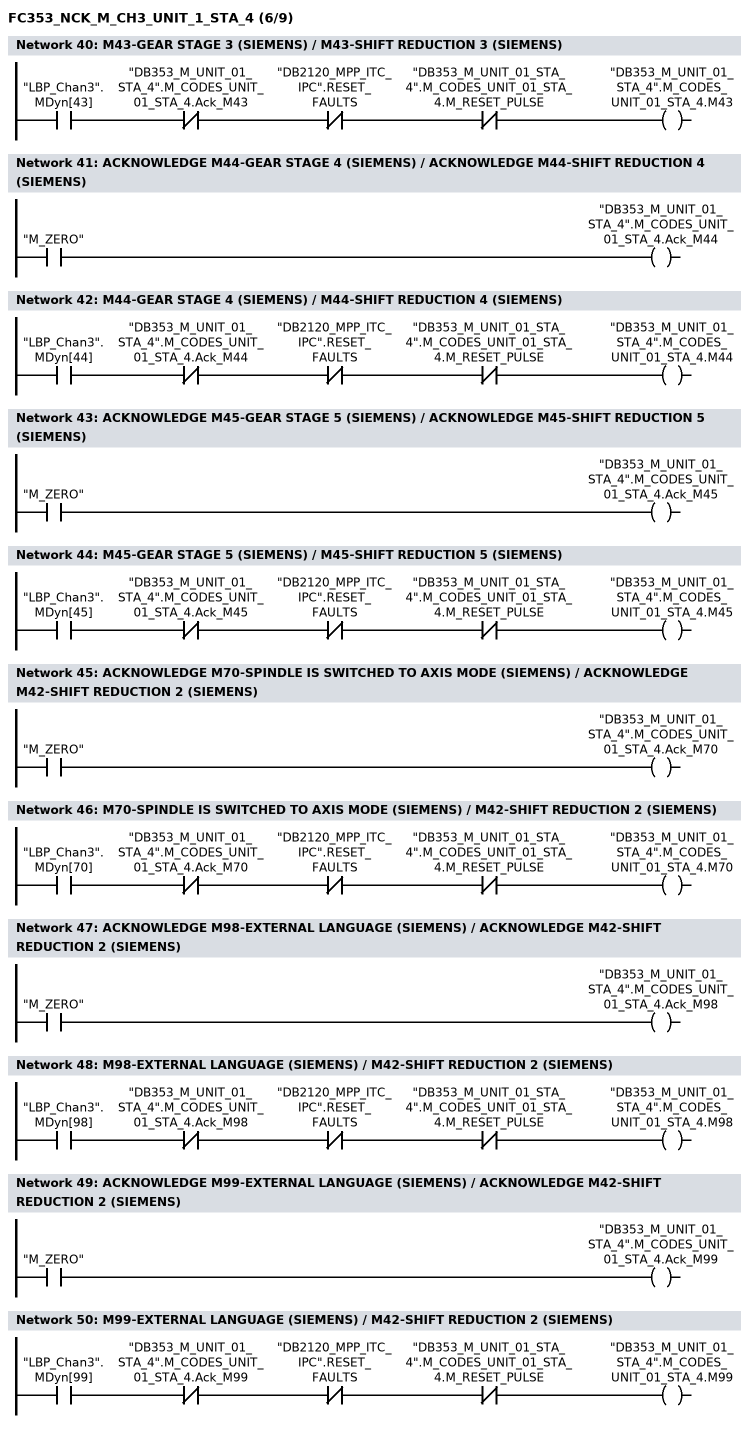
   RUNG wire#powerrail
      Contact( "LBP_Chan3".MDyn[43] )
      I_Contact( "DB353_M_UNIT_01_STA_4".M_CODES_UNIT_01_STA_4.Ack_M43 )
      I_Contact( "DB2120_MPP_ITC_IPC".RESET_FAULTS )
      I_Contact( "DB353_M_UNIT_01_STA_4".M_CODES_UNIT_01_STA_4.M_RESET_PULSE )
      Coil( "DB353_M_UNIT_01_STA_4".M_CODES_UNIT_01_STA_4.M43 )
   END_RUNG
   // the same network as SCL:
   "DB353_M_UNIT_01_STA_4".M_CODES_UNIT_01_STA_4.M43 := "LBP_Chan3".MDyn[43] AND NOT "DB353_M_UNIT_01_STA_4".M_CODES_UNIT_01_STA_4.Ack_M43 AND NOT "DB2120_MPP_ITC_IPC".RESET_FAULTS AND NOT "DB353_M_UNIT_01_STA_4".M_CODES_UNIT_01_STA_4.M_RESET_PULSE;
END_REGION

REGION Network 41: ACKNOWLEDGE M44-GEAR STAGE 4 (SIEMENS) / ACKNOWLEDGE M44-SHIFT REDUCTION 4 (SIEMENS)
   RUNG wire#powerrail
      Contact( "M_ZERO" )
      Coil( "DB353_M_UNIT_01_STA_4".M_CODES_UNIT_01_STA_4.Ack_M44 )
   END_RUNG
   // the same network as SCL:
   "DB353_M_UNIT_01_STA_4".M_CODES_UNIT_01_STA_4.Ack_M44 := "M_ZERO";
END_REGION

REGION Network 42: M44-GEAR STAGE 4 (SIEMENS) / M44-SHIFT REDUCTION 4 (SIEMENS)
   RUNG wire#powerrail
      Contact( "LBP_Chan3".MDyn[44] )
      I_Contact( "DB353_M_UNIT_01_STA_4".M_CODES_UNIT_01_STA_4.Ack_M44 )
      I_Contact( "DB2120_MPP_ITC_IPC".RESET_FAULTS )
      I_Contact( "DB353_M_UNIT_01_STA_4".M_CODES_UNIT_01_STA_4.M_RESET_PULSE )
      Coil( "DB353_M_UNIT_01_STA_4".M_CODES_UNIT_01_STA_4.M44 )
   END_RUNG
   // the same network as SCL:
   "DB353_M_UNIT_01_STA_4".M_CODES_UNIT_01_STA_4.M44 := "LBP_Chan3".MDyn[44] AND NOT "DB353_M_UNIT_01_STA_4".M_CODES_UNIT_01_STA_4.Ack_M44 AND NOT "DB2120_MPP_ITC_IPC".RESET_FAULTS AND NOT "DB353_M_UNIT_01_STA_4".M_CODES_UNIT_01_STA_4.M_RESET_PULSE;
END_REGION

REGION Network 43: ACKNOWLEDGE M45-GEAR STAGE 5 (SIEMENS) / ACKNOWLEDGE M45-SHIFT REDUCTION 5 (SIEMENS)
   RUNG wire#powerrail
      Contact( "M_ZERO" )
      Coil( "DB353_M_UNIT_01_STA_4".M_CODES_UNIT_01_STA_4.Ack_M45 )
   END_RUNG
   // the same network as SCL:
   "DB353_M_UNIT_01_STA_4".M_CODES_UNIT_01_STA_4.Ack_M45 := "M_ZERO";
END_REGION

REGION Network 44: M45-GEAR STAGE 5 (SIEMENS) / M45-SHIFT REDUCTION 5 (SIEMENS)
   RUNG wire#powerrail
      Contact( "LBP_Chan3".MDyn[45] )
      I_Contact( "DB353_M_UNIT_01_STA_4".M_CODES_UNIT_01_STA_4.Ack_M45 )
      I_Contact( "DB2120_MPP_ITC_IPC".RESET_FAULTS )
      I_Contact( "DB353_M_UNIT_01_STA_4".M_CODES_UNIT_01_STA_4.M_RESET_PULSE )
      Coil( "DB353_M_UNIT_01_STA_4".M_CODES_UNIT_01_STA_4.M45 )
   END_RUNG
   // the same network as SCL:
   "DB353_M_UNIT_01_STA_4".M_CODES_UNIT_01_STA_4.M45 := "LBP_Chan3".MDyn[45] AND NOT "DB353_M_UNIT_01_STA_4".M_CODES_UNIT_01_STA_4.Ack_M45 AND NOT "DB2120_MPP_ITC_IPC".RESET_FAULTS AND NOT "DB353_M_UNIT_01_STA_4".M_CODES_UNIT_01_STA_4.M_RESET_PULSE;
END_REGION

REGION Network 45: ACKNOWLEDGE M70-SPINDLE IS SWITCHED TO AXIS MODE (SIEMENS) / ACKNOWLEDGE M42-SHIFT REDUCTION 2 (SIEMENS)
   RUNG wire#powerrail
      Contact( "M_ZERO" )
      Coil( "DB353_M_UNIT_01_STA_4".M_CODES_UNIT_01_STA_4.Ack_M70 )
   END_RUNG
   // the same network as SCL:
   "DB353_M_UNIT_01_STA_4".M_CODES_UNIT_01_STA_4.Ack_M70 := "M_ZERO";
END_REGION

REGION Network 46: M70-SPINDLE IS SWITCHED TO AXIS MODE (SIEMENS) / M42-SHIFT REDUCTION 2 (SIEMENS)
   RUNG wire#powerrail
      Contact( "LBP_Chan3".MDyn[70] )
      I_Contact( "DB353_M_UNIT_01_STA_4".M_CODES_UNIT_01_STA_4.Ack_M70 )
      I_Contact( "DB2120_MPP_ITC_IPC".RESET_FAULTS )
      I_Contact( "DB353_M_UNIT_01_STA_4".M_CODES_UNIT_01_STA_4.M_RESET_PULSE )
      Coil( "DB353_M_UNIT_01_STA_4".M_CODES_UNIT_01_STA_4.M70 )
   END_RUNG
   // the same network as SCL:
   "DB353_M_UNIT_01_STA_4".M_CODES_UNIT_01_STA_4.M70 := "LBP_Chan3".MDyn[70] AND NOT "DB353_M_UNIT_01_STA_4".M_CODES_UNIT_01_STA_4.Ack_M70 AND NOT "DB2120_MPP_ITC_IPC".RESET_FAULTS AND NOT "DB353_M_UNIT_01_STA_4".M_CODES_UNIT_01_STA_4.M_RESET_PULSE;
END_REGION

REGION Network 47: ACKNOWLEDGE M98-EXTERNAL LANGUAGE (SIEMENS) / ACKNOWLEDGE M42-SHIFT REDUCTION 2 (SIEMENS)
   RUNG wire#powerrail
      Contact( "M_ZERO" )
      Coil( "DB353_M_UNIT_01_STA_4".M_CODES_UNIT_01_STA_4.Ack_M98 )
   END_RUNG
   // the same network as SCL:
   "DB353_M_UNIT_01_STA_4".M_CODES_UNIT_01_STA_4.Ack_M98 := "M_ZERO";
END_REGION

REGION Network 48: M98-EXTERNAL LANGUAGE (SIEMENS) / M42-SHIFT REDUCTION 2 (SIEMENS)
   RUNG wire#powerrail
      Contact( "LBP_Chan3".MDyn[98] )
      I_Contact( "DB353_M_UNIT_01_STA_4".M_CODES_UNIT_01_STA_4.Ack_M98 )
      I_Contact( "DB2120_MPP_ITC_IPC".RESET_FAULTS )
      I_Contact( "DB353_M_UNIT_01_STA_4".M_CODES_UNIT_01_STA_4.M_RESET_PULSE )
      Coil( "DB353_M_UNIT_01_STA_4".M_CODES_UNIT_01_STA_4.M98 )
   END_RUNG
   // the same network as SCL:
   "DB353_M_UNIT_01_STA_4".M_CODES_UNIT_01_STA_4.M98 := "LBP_Chan3".MDyn[98] AND NOT "DB353_M_UNIT_01_STA_4".M_CODES_UNIT_01_STA_4.Ack_M98 AND NOT "DB2120_MPP_ITC_IPC".RESET_FAULTS AND NOT "DB353_M_UNIT_01_STA_4".M_CODES_UNIT_01_STA_4.M_RESET_PULSE;
END_REGION

REGION Network 49: ACKNOWLEDGE M99-EXTERNAL LANGUAGE (SIEMENS) / ACKNOWLEDGE M42-SHIFT REDUCTION 2 (SIEMENS)
   RUNG wire#powerrail
      Contact( "M_ZERO" )
      Coil( "DB353_M_UNIT_01_STA_4".M_CODES_UNIT_01_STA_4.Ack_M99 )
   END_RUNG
   // the same network as SCL:
   "DB353_M_UNIT_01_STA_4".M_CODES_UNIT_01_STA_4.Ack_M99 := "M_ZERO";
END_REGION

REGION Network 50: M99-EXTERNAL LANGUAGE (SIEMENS) / M42-SHIFT REDUCTION 2 (SIEMENS)
   RUNG wire#powerrail
      Contact( "LBP_Chan3".MDyn[99] )
      I_Contact( "DB353_M_UNIT_01_STA_4".M_CODES_UNIT_01_STA_4.Ack_M99 )
      I_Contact( "DB2120_MPP_ITC_IPC".RESET_FAULTS )
      I_Contact( "DB353_M_UNIT_01_STA_4".M_CODES_UNIT_01_STA_4.M_RESET_PULSE )
      Coil( "DB353_M_UNIT_01_STA_4".M_CODES_UNIT_01_STA_4.M99 )
   END_RUNG
   // the same network as SCL:
   "DB353_M_UNIT_01_STA_4".M_CODES_UNIT_01_STA_4.M99 := "LBP_Chan3".MDyn[99] AND NOT "DB353_M_UNIT_01_STA_4".M_CODES_UNIT_01_STA_4.Ack_M99 AND NOT "DB2120_MPP_ITC_IPC".RESET_FAULTS AND NOT "DB353_M_UNIT_01_STA_4".M_CODES_UNIT_01_STA_4.M_RESET_PULSE;
END_REGION

REGION Network 51: ACKNOWLEDGE M100-WAIT UNTIL E AXIS IN POSITION FIXTURE 1 STATION 4(READ-IN DISABLE) / ACKNOWLEDGE M23-SWITCH ON SPINDLE FRAME BLOWING
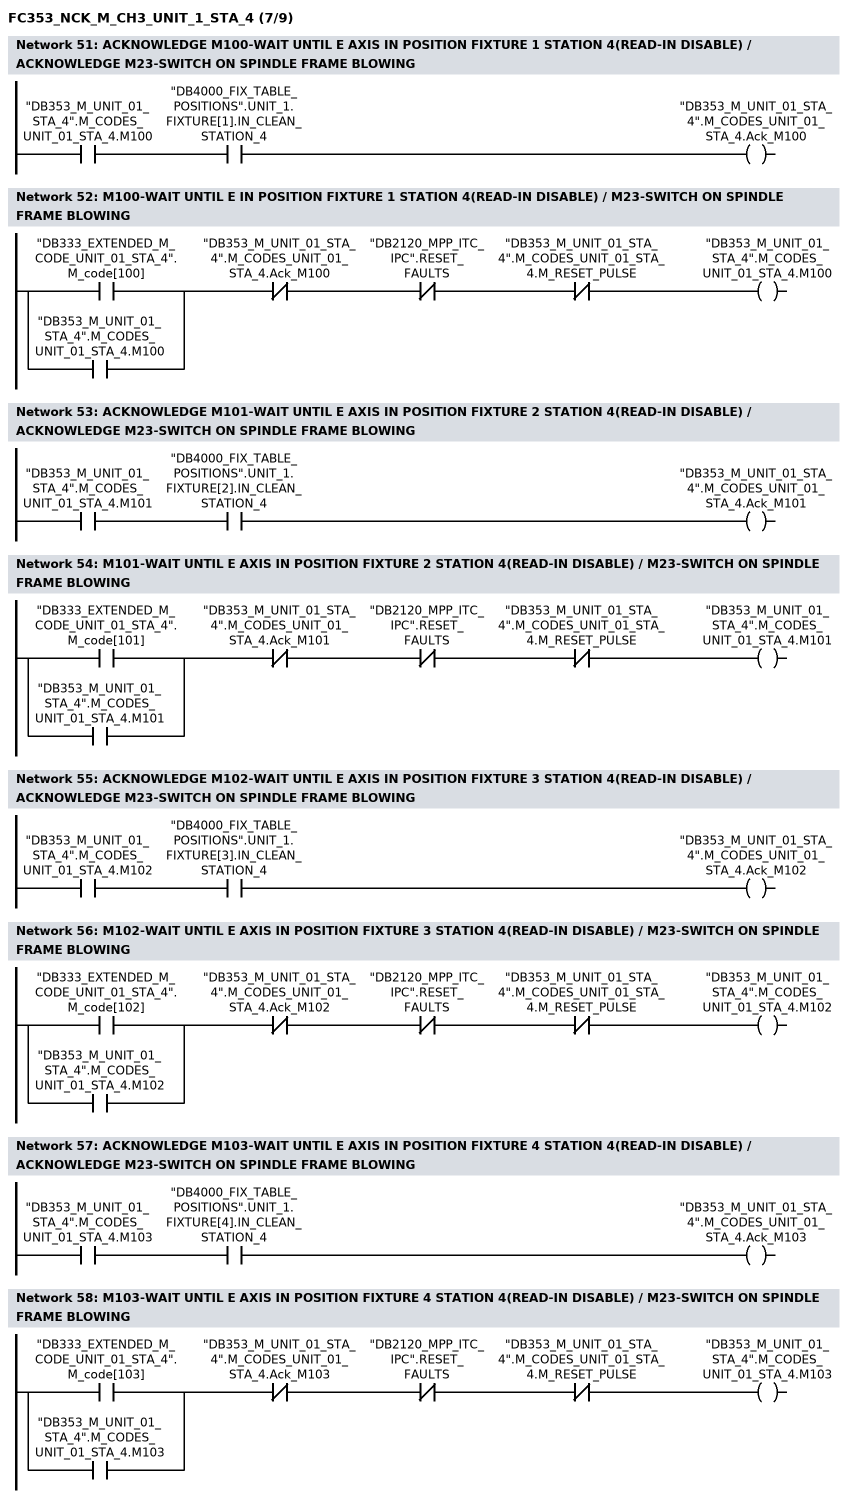
   RUNG wire#powerrail
      Contact( "DB353_M_UNIT_01_STA_4".M_CODES_UNIT_01_STA_4.M100 )
      Contact( "DB4000_FIX_TABLE_POSITIONS".UNIT_1.FIXTURE[1].IN_CLEAN_STATION_4 )
      Coil( "DB353_M_UNIT_01_STA_4".M_CODES_UNIT_01_STA_4.Ack_M100 )
   END_RUNG
   // the same network as SCL:
   "DB353_M_UNIT_01_STA_4".M_CODES_UNIT_01_STA_4.Ack_M100 := "DB353_M_UNIT_01_STA_4".M_CODES_UNIT_01_STA_4.M100 AND "DB4000_FIX_TABLE_POSITIONS".UNIT_1.FIXTURE[1].IN_CLEAN_STATION_4;
END_REGION

REGION Network 52: M100-WAIT UNTIL E IN POSITION FIXTURE 1 STATION 4(READ-IN DISABLE) / M23-SWITCH ON SPINDLE FRAME BLOWING
   RUNG wire#powerrail
      Contact( "DB333_EXTENDED_M_CODE_UNIT_01_STA_4".M_code[100] )
      wire#w1
      I_Contact( "DB353_M_UNIT_01_STA_4".M_CODES_UNIT_01_STA_4.Ack_M100 )
      I_Contact( "DB2120_MPP_ITC_IPC".RESET_FAULTS )
      I_Contact( "DB353_M_UNIT_01_STA_4".M_CODES_UNIT_01_STA_4.M_RESET_PULSE )
      Coil( "DB353_M_UNIT_01_STA_4".M_CODES_UNIT_01_STA_4.M100 )
   END_RUNG
   RUNG wire#powerrail
      Contact( "DB353_M_UNIT_01_STA_4".M_CODES_UNIT_01_STA_4.M100 )
   END_RUNG wire#w1
   // the same network as SCL:
   "DB353_M_UNIT_01_STA_4".M_CODES_UNIT_01_STA_4.M100 := ("DB333_EXTENDED_M_CODE_UNIT_01_STA_4".M_code[100] OR "DB353_M_UNIT_01_STA_4".M_CODES_UNIT_01_STA_4.M100) AND NOT "DB353_M_UNIT_01_STA_4".M_CODES_UNIT_01_STA_4.Ack_M100 AND NOT "DB2120_MPP_ITC_IPC".RESET_FAULTS AND NOT "DB353_M_UNIT_01_STA_4".M_CODES_UNIT_01_STA_4.M_RESET_PULSE;
END_REGION

REGION Network 53: ACKNOWLEDGE M101-WAIT UNTIL E AXIS IN POSITION FIXTURE 2 STATION 4(READ-IN DISABLE) / ACKNOWLEDGE M23-SWITCH ON SPINDLE FRAME BLOWING
   RUNG wire#powerrail
      Contact( "DB353_M_UNIT_01_STA_4".M_CODES_UNIT_01_STA_4.M101 )
      Contact( "DB4000_FIX_TABLE_POSITIONS".UNIT_1.FIXTURE[2].IN_CLEAN_STATION_4 )
      Coil( "DB353_M_UNIT_01_STA_4".M_CODES_UNIT_01_STA_4.Ack_M101 )
   END_RUNG
   // the same network as SCL:
   "DB353_M_UNIT_01_STA_4".M_CODES_UNIT_01_STA_4.Ack_M101 := "DB353_M_UNIT_01_STA_4".M_CODES_UNIT_01_STA_4.M101 AND "DB4000_FIX_TABLE_POSITIONS".UNIT_1.FIXTURE[2].IN_CLEAN_STATION_4;
END_REGION

REGION Network 54: M101-WAIT UNTIL E AXIS IN POSITION FIXTURE 2 STATION 4(READ-IN DISABLE) / M23-SWITCH ON SPINDLE FRAME BLOWING
   RUNG wire#powerrail
      Contact( "DB333_EXTENDED_M_CODE_UNIT_01_STA_4".M_code[101] )
      wire#w1
      I_Contact( "DB353_M_UNIT_01_STA_4".M_CODES_UNIT_01_STA_4.Ack_M101 )
      I_Contact( "DB2120_MPP_ITC_IPC".RESET_FAULTS )
      I_Contact( "DB353_M_UNIT_01_STA_4".M_CODES_UNIT_01_STA_4.M_RESET_PULSE )
      Coil( "DB353_M_UNIT_01_STA_4".M_CODES_UNIT_01_STA_4.M101 )
   END_RUNG
   RUNG wire#powerrail
      Contact( "DB353_M_UNIT_01_STA_4".M_CODES_UNIT_01_STA_4.M101 )
   END_RUNG wire#w1
   // the same network as SCL:
   "DB353_M_UNIT_01_STA_4".M_CODES_UNIT_01_STA_4.M101 := ("DB333_EXTENDED_M_CODE_UNIT_01_STA_4".M_code[101] OR "DB353_M_UNIT_01_STA_4".M_CODES_UNIT_01_STA_4.M101) AND NOT "DB353_M_UNIT_01_STA_4".M_CODES_UNIT_01_STA_4.Ack_M101 AND NOT "DB2120_MPP_ITC_IPC".RESET_FAULTS AND NOT "DB353_M_UNIT_01_STA_4".M_CODES_UNIT_01_STA_4.M_RESET_PULSE;
END_REGION

REGION Network 55: ACKNOWLEDGE M102-WAIT UNTIL E AXIS IN POSITION FIXTURE 3 STATION 4(READ-IN DISABLE) / ACKNOWLEDGE M23-SWITCH ON SPINDLE FRAME BLOWING
   RUNG wire#powerrail
      Contact( "DB353_M_UNIT_01_STA_4".M_CODES_UNIT_01_STA_4.M102 )
      Contact( "DB4000_FIX_TABLE_POSITIONS".UNIT_1.FIXTURE[3].IN_CLEAN_STATION_4 )
      Coil( "DB353_M_UNIT_01_STA_4".M_CODES_UNIT_01_STA_4.Ack_M102 )
   END_RUNG
   // the same network as SCL:
   "DB353_M_UNIT_01_STA_4".M_CODES_UNIT_01_STA_4.Ack_M102 := "DB353_M_UNIT_01_STA_4".M_CODES_UNIT_01_STA_4.M102 AND "DB4000_FIX_TABLE_POSITIONS".UNIT_1.FIXTURE[3].IN_CLEAN_STATION_4;
END_REGION

REGION Network 56: M102-WAIT UNTIL E AXIS IN POSITION FIXTURE 3 STATION 4(READ-IN DISABLE) / M23-SWITCH ON SPINDLE FRAME BLOWING
   RUNG wire#powerrail
      Contact( "DB333_EXTENDED_M_CODE_UNIT_01_STA_4".M_code[102] )
      wire#w1
      I_Contact( "DB353_M_UNIT_01_STA_4".M_CODES_UNIT_01_STA_4.Ack_M102 )
      I_Contact( "DB2120_MPP_ITC_IPC".RESET_FAULTS )
      I_Contact( "DB353_M_UNIT_01_STA_4".M_CODES_UNIT_01_STA_4.M_RESET_PULSE )
      Coil( "DB353_M_UNIT_01_STA_4".M_CODES_UNIT_01_STA_4.M102 )
   END_RUNG
   RUNG wire#powerrail
      Contact( "DB353_M_UNIT_01_STA_4".M_CODES_UNIT_01_STA_4.M102 )
   END_RUNG wire#w1
   // the same network as SCL:
   "DB353_M_UNIT_01_STA_4".M_CODES_UNIT_01_STA_4.M102 := ("DB333_EXTENDED_M_CODE_UNIT_01_STA_4".M_code[102] OR "DB353_M_UNIT_01_STA_4".M_CODES_UNIT_01_STA_4.M102) AND NOT "DB353_M_UNIT_01_STA_4".M_CODES_UNIT_01_STA_4.Ack_M102 AND NOT "DB2120_MPP_ITC_IPC".RESET_FAULTS AND NOT "DB353_M_UNIT_01_STA_4".M_CODES_UNIT_01_STA_4.M_RESET_PULSE;
END_REGION

REGION Network 57: ACKNOWLEDGE M103-WAIT UNTIL E AXIS IN POSITION FIXTURE 4 STATION 4(READ-IN DISABLE) / ACKNOWLEDGE M23-SWITCH ON SPINDLE FRAME BLOWING
   RUNG wire#powerrail
      Contact( "DB353_M_UNIT_01_STA_4".M_CODES_UNIT_01_STA_4.M103 )
      Contact( "DB4000_FIX_TABLE_POSITIONS".UNIT_1.FIXTURE[4].IN_CLEAN_STATION_4 )
      Coil( "DB353_M_UNIT_01_STA_4".M_CODES_UNIT_01_STA_4.Ack_M103 )
   END_RUNG
   // the same network as SCL:
   "DB353_M_UNIT_01_STA_4".M_CODES_UNIT_01_STA_4.Ack_M103 := "DB353_M_UNIT_01_STA_4".M_CODES_UNIT_01_STA_4.M103 AND "DB4000_FIX_TABLE_POSITIONS".UNIT_1.FIXTURE[4].IN_CLEAN_STATION_4;
END_REGION

REGION Network 58: M103-WAIT UNTIL E AXIS IN POSITION FIXTURE 4 STATION 4(READ-IN DISABLE) / M23-SWITCH ON SPINDLE FRAME BLOWING
   RUNG wire#powerrail
      Contact( "DB333_EXTENDED_M_CODE_UNIT_01_STA_4".M_code[103] )
      wire#w1
      I_Contact( "DB353_M_UNIT_01_STA_4".M_CODES_UNIT_01_STA_4.Ack_M103 )
      I_Contact( "DB2120_MPP_ITC_IPC".RESET_FAULTS )
      I_Contact( "DB353_M_UNIT_01_STA_4".M_CODES_UNIT_01_STA_4.M_RESET_PULSE )
      Coil( "DB353_M_UNIT_01_STA_4".M_CODES_UNIT_01_STA_4.M103 )
   END_RUNG
   RUNG wire#powerrail
      Contact( "DB353_M_UNIT_01_STA_4".M_CODES_UNIT_01_STA_4.M103 )
   END_RUNG wire#w1
   // the same network as SCL:
   "DB353_M_UNIT_01_STA_4".M_CODES_UNIT_01_STA_4.M103 := ("DB333_EXTENDED_M_CODE_UNIT_01_STA_4".M_code[103] OR "DB353_M_UNIT_01_STA_4".M_CODES_UNIT_01_STA_4.M103) AND NOT "DB353_M_UNIT_01_STA_4".M_CODES_UNIT_01_STA_4.Ack_M103 AND NOT "DB2120_MPP_ITC_IPC".RESET_FAULTS AND NOT "DB353_M_UNIT_01_STA_4".M_CODES_UNIT_01_STA_4.M_RESET_PULSE;
END_REGION

REGION Network 59: ACKNOWLEDGE M110-UNBLOCK TABLE
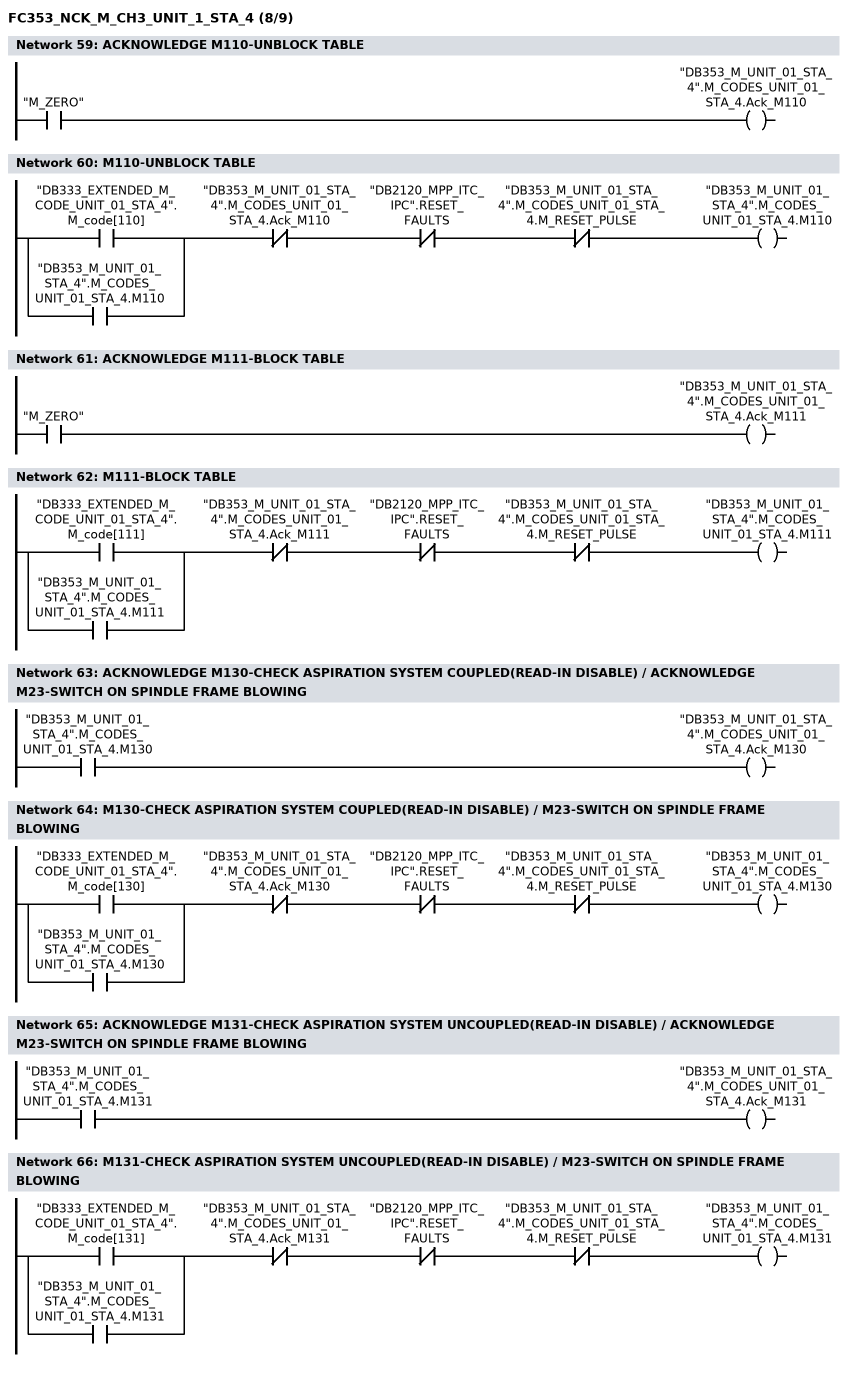
   RUNG wire#powerrail
      Contact( "M_ZERO" )
      Coil( "DB353_M_UNIT_01_STA_4".M_CODES_UNIT_01_STA_4.Ack_M110 )
   END_RUNG
   // the same network as SCL:
   "DB353_M_UNIT_01_STA_4".M_CODES_UNIT_01_STA_4.Ack_M110 := "M_ZERO";
END_REGION

REGION Network 60: M110-UNBLOCK TABLE
   RUNG wire#powerrail
      Contact( "DB333_EXTENDED_M_CODE_UNIT_01_STA_4".M_code[110] )
      wire#w1
      I_Contact( "DB353_M_UNIT_01_STA_4".M_CODES_UNIT_01_STA_4.Ack_M110 )
      I_Contact( "DB2120_MPP_ITC_IPC".RESET_FAULTS )
      I_Contact( "DB353_M_UNIT_01_STA_4".M_CODES_UNIT_01_STA_4.M_RESET_PULSE )
      Coil( "DB353_M_UNIT_01_STA_4".M_CODES_UNIT_01_STA_4.M110 )
   END_RUNG
   RUNG wire#powerrail
      Contact( "DB353_M_UNIT_01_STA_4".M_CODES_UNIT_01_STA_4.M110 )
   END_RUNG wire#w1
   // the same network as SCL:
   "DB353_M_UNIT_01_STA_4".M_CODES_UNIT_01_STA_4.M110 := ("DB333_EXTENDED_M_CODE_UNIT_01_STA_4".M_code[110] OR "DB353_M_UNIT_01_STA_4".M_CODES_UNIT_01_STA_4.M110) AND NOT "DB353_M_UNIT_01_STA_4".M_CODES_UNIT_01_STA_4.Ack_M110 AND NOT "DB2120_MPP_ITC_IPC".RESET_FAULTS AND NOT "DB353_M_UNIT_01_STA_4".M_CODES_UNIT_01_STA_4.M_RESET_PULSE;
END_REGION

REGION Network 61: ACKNOWLEDGE M111-BLOCK TABLE
   RUNG wire#powerrail
      Contact( "M_ZERO" )
      Coil( "DB353_M_UNIT_01_STA_4".M_CODES_UNIT_01_STA_4.Ack_M111 )
   END_RUNG
   // the same network as SCL:
   "DB353_M_UNIT_01_STA_4".M_CODES_UNIT_01_STA_4.Ack_M111 := "M_ZERO";
END_REGION

REGION Network 62: M111-BLOCK TABLE
   RUNG wire#powerrail
      Contact( "DB333_EXTENDED_M_CODE_UNIT_01_STA_4".M_code[111] )
      wire#w1
      I_Contact( "DB353_M_UNIT_01_STA_4".M_CODES_UNIT_01_STA_4.Ack_M111 )
      I_Contact( "DB2120_MPP_ITC_IPC".RESET_FAULTS )
      I_Contact( "DB353_M_UNIT_01_STA_4".M_CODES_UNIT_01_STA_4.M_RESET_PULSE )
      Coil( "DB353_M_UNIT_01_STA_4".M_CODES_UNIT_01_STA_4.M111 )
   END_RUNG
   RUNG wire#powerrail
      Contact( "DB353_M_UNIT_01_STA_4".M_CODES_UNIT_01_STA_4.M111 )
   END_RUNG wire#w1
   // the same network as SCL:
   "DB353_M_UNIT_01_STA_4".M_CODES_UNIT_01_STA_4.M111 := ("DB333_EXTENDED_M_CODE_UNIT_01_STA_4".M_code[111] OR "DB353_M_UNIT_01_STA_4".M_CODES_UNIT_01_STA_4.M111) AND NOT "DB353_M_UNIT_01_STA_4".M_CODES_UNIT_01_STA_4.Ack_M111 AND NOT "DB2120_MPP_ITC_IPC".RESET_FAULTS AND NOT "DB353_M_UNIT_01_STA_4".M_CODES_UNIT_01_STA_4.M_RESET_PULSE;
END_REGION

REGION Network 63: ACKNOWLEDGE M130-CHECK ASPIRATION SYSTEM COUPLED(READ-IN DISABLE) / ACKNOWLEDGE M23-SWITCH ON SPINDLE FRAME BLOWING
   RUNG wire#powerrail
      Contact( "DB353_M_UNIT_01_STA_4".M_CODES_UNIT_01_STA_4.M130 )
      Coil( "DB353_M_UNIT_01_STA_4".M_CODES_UNIT_01_STA_4.Ack_M130 )
   END_RUNG
   // the same network as SCL:
   "DB353_M_UNIT_01_STA_4".M_CODES_UNIT_01_STA_4.Ack_M130 := "DB353_M_UNIT_01_STA_4".M_CODES_UNIT_01_STA_4.M130;
END_REGION

REGION Network 64: M130-CHECK ASPIRATION SYSTEM COUPLED(READ-IN DISABLE) / M23-SWITCH ON SPINDLE FRAME BLOWING
   RUNG wire#powerrail
      Contact( "DB333_EXTENDED_M_CODE_UNIT_01_STA_4".M_code[130] )
      wire#w1
      I_Contact( "DB353_M_UNIT_01_STA_4".M_CODES_UNIT_01_STA_4.Ack_M130 )
      I_Contact( "DB2120_MPP_ITC_IPC".RESET_FAULTS )
      I_Contact( "DB353_M_UNIT_01_STA_4".M_CODES_UNIT_01_STA_4.M_RESET_PULSE )
      Coil( "DB353_M_UNIT_01_STA_4".M_CODES_UNIT_01_STA_4.M130 )
   END_RUNG
   RUNG wire#powerrail
      Contact( "DB353_M_UNIT_01_STA_4".M_CODES_UNIT_01_STA_4.M130 )
   END_RUNG wire#w1
   // the same network as SCL:
   "DB353_M_UNIT_01_STA_4".M_CODES_UNIT_01_STA_4.M130 := ("DB333_EXTENDED_M_CODE_UNIT_01_STA_4".M_code[130] OR "DB353_M_UNIT_01_STA_4".M_CODES_UNIT_01_STA_4.M130) AND NOT "DB353_M_UNIT_01_STA_4".M_CODES_UNIT_01_STA_4.Ack_M130 AND NOT "DB2120_MPP_ITC_IPC".RESET_FAULTS AND NOT "DB353_M_UNIT_01_STA_4".M_CODES_UNIT_01_STA_4.M_RESET_PULSE;
END_REGION

REGION Network 65: ACKNOWLEDGE M131-CHECK ASPIRATION SYSTEM UNCOUPLED(READ-IN DISABLE) / ACKNOWLEDGE M23-SWITCH ON SPINDLE FRAME BLOWING
   RUNG wire#powerrail
      Contact( "DB353_M_UNIT_01_STA_4".M_CODES_UNIT_01_STA_4.M131 )
      Coil( "DB353_M_UNIT_01_STA_4".M_CODES_UNIT_01_STA_4.Ack_M131 )
   END_RUNG
   // the same network as SCL:
   "DB353_M_UNIT_01_STA_4".M_CODES_UNIT_01_STA_4.Ack_M131 := "DB353_M_UNIT_01_STA_4".M_CODES_UNIT_01_STA_4.M131;
END_REGION

REGION Network 66: M131-CHECK ASPIRATION SYSTEM UNCOUPLED(READ-IN DISABLE) / M23-SWITCH ON SPINDLE FRAME BLOWING
   RUNG wire#powerrail
      Contact( "DB333_EXTENDED_M_CODE_UNIT_01_STA_4".M_code[131] )
      wire#w1
      I_Contact( "DB353_M_UNIT_01_STA_4".M_CODES_UNIT_01_STA_4.Ack_M131 )
      I_Contact( "DB2120_MPP_ITC_IPC".RESET_FAULTS )
      I_Contact( "DB353_M_UNIT_01_STA_4".M_CODES_UNIT_01_STA_4.M_RESET_PULSE )
      Coil( "DB353_M_UNIT_01_STA_4".M_CODES_UNIT_01_STA_4.M131 )
   END_RUNG
   RUNG wire#powerrail
      Contact( "DB353_M_UNIT_01_STA_4".M_CODES_UNIT_01_STA_4.M131 )
   END_RUNG wire#w1
   // the same network as SCL:
   "DB353_M_UNIT_01_STA_4".M_CODES_UNIT_01_STA_4.M131 := ("DB333_EXTENDED_M_CODE_UNIT_01_STA_4".M_code[131] OR "DB353_M_UNIT_01_STA_4".M_CODES_UNIT_01_STA_4.M131) AND NOT "DB353_M_UNIT_01_STA_4".M_CODES_UNIT_01_STA_4.Ack_M131 AND NOT "DB2120_MPP_ITC_IPC".RESET_FAULTS AND NOT "DB353_M_UNIT_01_STA_4".M_CODES_UNIT_01_STA_4.M_RESET_PULSE;
END_REGION

REGION Network 67: ACKNOWLEDGE M138-CLEANING VALVE SWITCH ON STATION 4 / ACKNOWLEDGE M23-SWITCH ON SPINDLE FRAME BLOWING
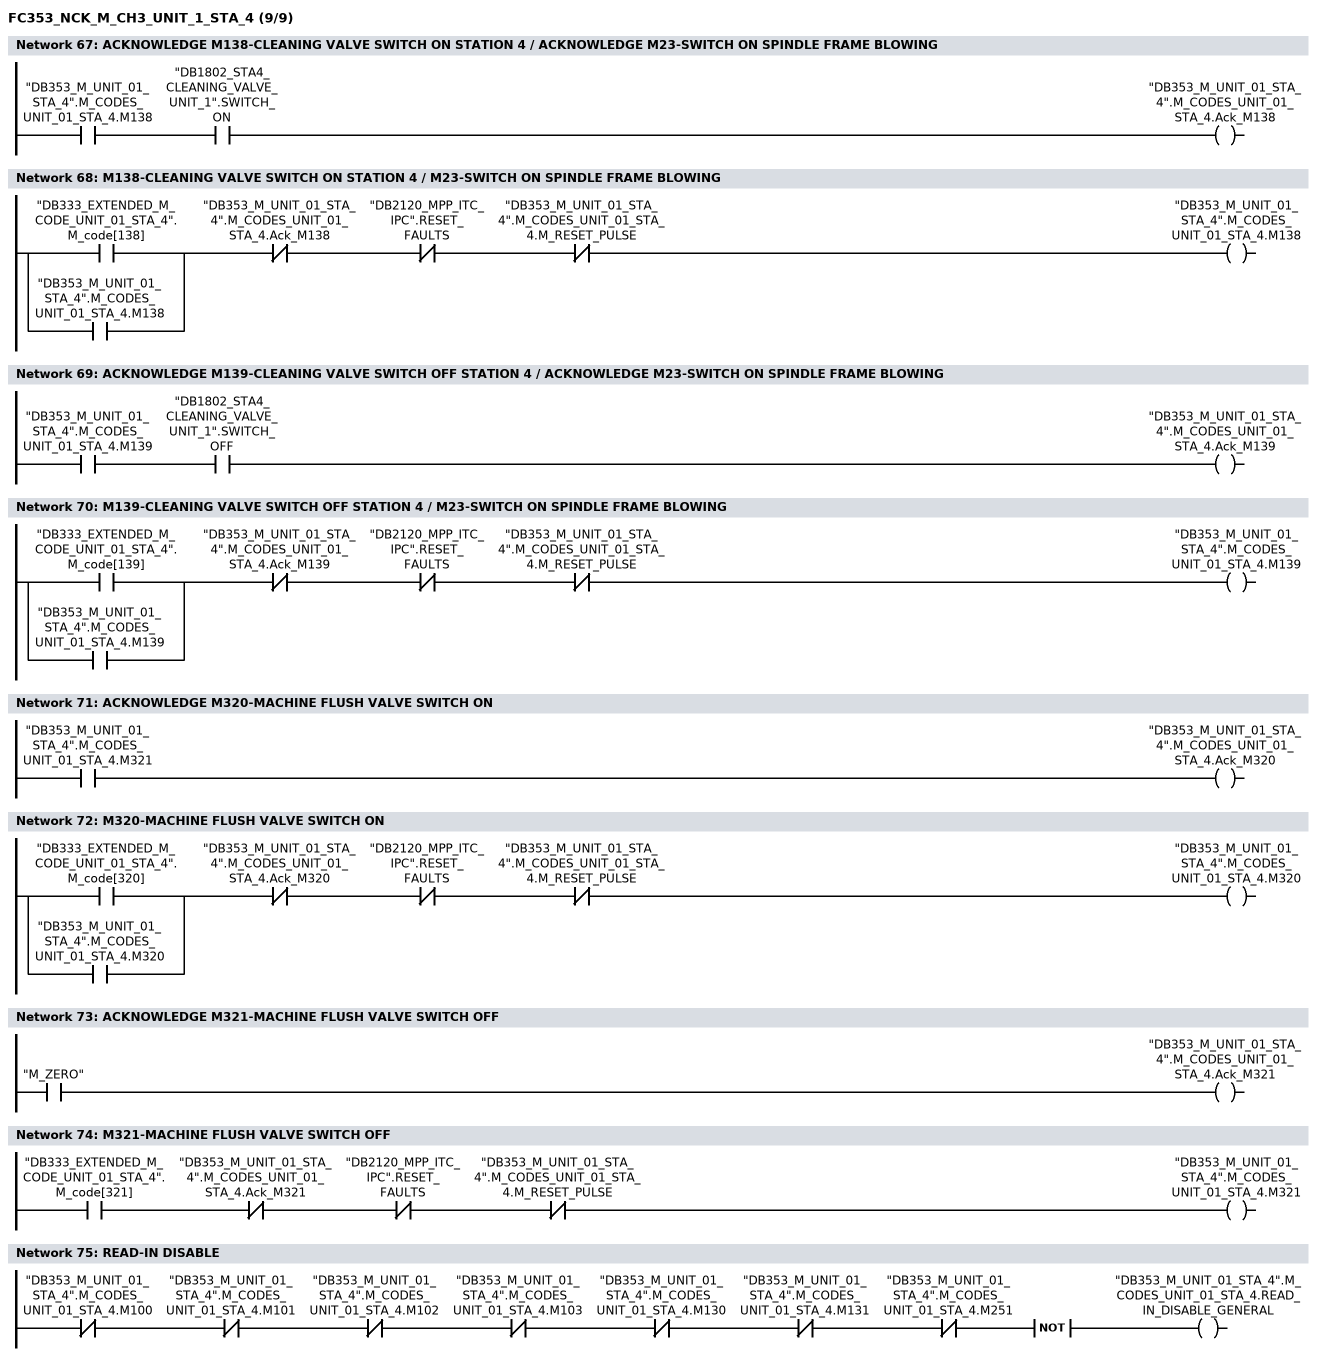
   RUNG wire#powerrail
      Contact( "DB353_M_UNIT_01_STA_4".M_CODES_UNIT_01_STA_4.M138 )
      Contact( "DB1802_STA4_CLEANING_VALVE_UNIT_1".SWITCH_ON )
      Coil( "DB353_M_UNIT_01_STA_4".M_CODES_UNIT_01_STA_4.Ack_M138 )
   END_RUNG
   // the same network as SCL:
   "DB353_M_UNIT_01_STA_4".M_CODES_UNIT_01_STA_4.Ack_M138 := "DB353_M_UNIT_01_STA_4".M_CODES_UNIT_01_STA_4.M138 AND "DB1802_STA4_CLEANING_VALVE_UNIT_1".SWITCH_ON;
END_REGION

REGION Network 68: M138-CLEANING VALVE SWITCH ON STATION 4 / M23-SWITCH ON SPINDLE FRAME BLOWING
   RUNG wire#powerrail
      Contact( "DB333_EXTENDED_M_CODE_UNIT_01_STA_4".M_code[138] )
      wire#w1
      I_Contact( "DB353_M_UNIT_01_STA_4".M_CODES_UNIT_01_STA_4.Ack_M138 )
      I_Contact( "DB2120_MPP_ITC_IPC".RESET_FAULTS )
      I_Contact( "DB353_M_UNIT_01_STA_4".M_CODES_UNIT_01_STA_4.M_RESET_PULSE )
      Coil( "DB353_M_UNIT_01_STA_4".M_CODES_UNIT_01_STA_4.M138 )
   END_RUNG
   RUNG wire#powerrail
      Contact( "DB353_M_UNIT_01_STA_4".M_CODES_UNIT_01_STA_4.M138 )
   END_RUNG wire#w1
   // the same network as SCL:
   "DB353_M_UNIT_01_STA_4".M_CODES_UNIT_01_STA_4.M138 := ("DB333_EXTENDED_M_CODE_UNIT_01_STA_4".M_code[138] OR "DB353_M_UNIT_01_STA_4".M_CODES_UNIT_01_STA_4.M138) AND NOT "DB353_M_UNIT_01_STA_4".M_CODES_UNIT_01_STA_4.Ack_M138 AND NOT "DB2120_MPP_ITC_IPC".RESET_FAULTS AND NOT "DB353_M_UNIT_01_STA_4".M_CODES_UNIT_01_STA_4.M_RESET_PULSE;
END_REGION

REGION Network 69: ACKNOWLEDGE M139-CLEANING VALVE SWITCH OFF STATION 4 / ACKNOWLEDGE M23-SWITCH ON SPINDLE FRAME BLOWING
   RUNG wire#powerrail
      Contact( "DB353_M_UNIT_01_STA_4".M_CODES_UNIT_01_STA_4.M139 )
      Contact( "DB1802_STA4_CLEANING_VALVE_UNIT_1".SWITCH_OFF )
      Coil( "DB353_M_UNIT_01_STA_4".M_CODES_UNIT_01_STA_4.Ack_M139 )
   END_RUNG
   // the same network as SCL:
   "DB353_M_UNIT_01_STA_4".M_CODES_UNIT_01_STA_4.Ack_M139 := "DB353_M_UNIT_01_STA_4".M_CODES_UNIT_01_STA_4.M139 AND "DB1802_STA4_CLEANING_VALVE_UNIT_1".SWITCH_OFF;
END_REGION

REGION Network 70: M139-CLEANING VALVE SWITCH OFF STATION 4 / M23-SWITCH ON SPINDLE FRAME BLOWING
   RUNG wire#powerrail
      Contact( "DB333_EXTENDED_M_CODE_UNIT_01_STA_4".M_code[139] )
      wire#w1
      I_Contact( "DB353_M_UNIT_01_STA_4".M_CODES_UNIT_01_STA_4.Ack_M139 )
      I_Contact( "DB2120_MPP_ITC_IPC".RESET_FAULTS )
      I_Contact( "DB353_M_UNIT_01_STA_4".M_CODES_UNIT_01_STA_4.M_RESET_PULSE )
      Coil( "DB353_M_UNIT_01_STA_4".M_CODES_UNIT_01_STA_4.M139 )
   END_RUNG
   RUNG wire#powerrail
      Contact( "DB353_M_UNIT_01_STA_4".M_CODES_UNIT_01_STA_4.M139 )
   END_RUNG wire#w1
   // the same network as SCL:
   "DB353_M_UNIT_01_STA_4".M_CODES_UNIT_01_STA_4.M139 := ("DB333_EXTENDED_M_CODE_UNIT_01_STA_4".M_code[139] OR "DB353_M_UNIT_01_STA_4".M_CODES_UNIT_01_STA_4.M139) AND NOT "DB353_M_UNIT_01_STA_4".M_CODES_UNIT_01_STA_4.Ack_M139 AND NOT "DB2120_MPP_ITC_IPC".RESET_FAULTS AND NOT "DB353_M_UNIT_01_STA_4".M_CODES_UNIT_01_STA_4.M_RESET_PULSE;
END_REGION

REGION Network 71: ACKNOWLEDGE M320-MACHINE FLUSH VALVE SWITCH ON
   RUNG wire#powerrail
      Contact( "DB353_M_UNIT_01_STA_4".M_CODES_UNIT_01_STA_4.M321 )
      Coil( "DB353_M_UNIT_01_STA_4".M_CODES_UNIT_01_STA_4.Ack_M320 )
   END_RUNG
   // the same network as SCL:
   "DB353_M_UNIT_01_STA_4".M_CODES_UNIT_01_STA_4.Ack_M320 := "DB353_M_UNIT_01_STA_4".M_CODES_UNIT_01_STA_4.M321;
END_REGION

REGION Network 72: M320-MACHINE FLUSH VALVE SWITCH ON
   RUNG wire#powerrail
      Contact( "DB333_EXTENDED_M_CODE_UNIT_01_STA_4".M_code[320] )
      wire#w1
      I_Contact( "DB353_M_UNIT_01_STA_4".M_CODES_UNIT_01_STA_4.Ack_M320 )
      I_Contact( "DB2120_MPP_ITC_IPC".RESET_FAULTS )
      I_Contact( "DB353_M_UNIT_01_STA_4".M_CODES_UNIT_01_STA_4.M_RESET_PULSE )
      Coil( "DB353_M_UNIT_01_STA_4".M_CODES_UNIT_01_STA_4.M320 )
   END_RUNG
   RUNG wire#powerrail
      Contact( "DB353_M_UNIT_01_STA_4".M_CODES_UNIT_01_STA_4.M320 )
   END_RUNG wire#w1
   // the same network as SCL:
   "DB353_M_UNIT_01_STA_4".M_CODES_UNIT_01_STA_4.M320 := ("DB333_EXTENDED_M_CODE_UNIT_01_STA_4".M_code[320] OR "DB353_M_UNIT_01_STA_4".M_CODES_UNIT_01_STA_4.M320) AND NOT "DB353_M_UNIT_01_STA_4".M_CODES_UNIT_01_STA_4.Ack_M320 AND NOT "DB2120_MPP_ITC_IPC".RESET_FAULTS AND NOT "DB353_M_UNIT_01_STA_4".M_CODES_UNIT_01_STA_4.M_RESET_PULSE;
END_REGION

REGION Network 73: ACKNOWLEDGE M321-MACHINE FLUSH VALVE SWITCH OFF
   RUNG wire#powerrail
      Contact( "M_ZERO" )
      Coil( "DB353_M_UNIT_01_STA_4".M_CODES_UNIT_01_STA_4.Ack_M321 )
   END_RUNG
   // the same network as SCL:
   "DB353_M_UNIT_01_STA_4".M_CODES_UNIT_01_STA_4.Ack_M321 := "M_ZERO";
END_REGION

REGION Network 74: M321-MACHINE FLUSH VALVE SWITCH OFF
   RUNG wire#powerrail
      Contact( "DB333_EXTENDED_M_CODE_UNIT_01_STA_4".M_code[321] )
      I_Contact( "DB353_M_UNIT_01_STA_4".M_CODES_UNIT_01_STA_4.Ack_M321 )
      I_Contact( "DB2120_MPP_ITC_IPC".RESET_FAULTS )
      I_Contact( "DB353_M_UNIT_01_STA_4".M_CODES_UNIT_01_STA_4.M_RESET_PULSE )
      Coil( "DB353_M_UNIT_01_STA_4".M_CODES_UNIT_01_STA_4.M321 )
   END_RUNG
   // the same network as SCL:
   "DB353_M_UNIT_01_STA_4".M_CODES_UNIT_01_STA_4.M321 := "DB333_EXTENDED_M_CODE_UNIT_01_STA_4".M_code[321] AND NOT "DB353_M_UNIT_01_STA_4".M_CODES_UNIT_01_STA_4.Ack_M321 AND NOT "DB2120_MPP_ITC_IPC".RESET_FAULTS AND NOT "DB353_M_UNIT_01_STA_4".M_CODES_UNIT_01_STA_4.M_RESET_PULSE;
END_REGION

REGION Network 75: READ-IN DISABLE
   RUNG wire#powerrail
      I_Contact( "DB353_M_UNIT_01_STA_4".M_CODES_UNIT_01_STA_4.M100 )
      I_Contact( "DB353_M_UNIT_01_STA_4".M_CODES_UNIT_01_STA_4.M101 )
      I_Contact( "DB353_M_UNIT_01_STA_4".M_CODES_UNIT_01_STA_4.M102 )
      I_Contact( "DB353_M_UNIT_01_STA_4".M_CODES_UNIT_01_STA_4.M103 )
      I_Contact( "DB353_M_UNIT_01_STA_4".M_CODES_UNIT_01_STA_4.M130 )
      I_Contact( "DB353_M_UNIT_01_STA_4".M_CODES_UNIT_01_STA_4.M131 )
      I_Contact( "DB353_M_UNIT_01_STA_4".M_CODES_UNIT_01_STA_4.M251 )
      Not()
      Coil( "DB353_M_UNIT_01_STA_4".M_CODES_UNIT_01_STA_4.READ_IN_DISABLE_GENERAL )
   END_RUNG
   // the same network as SCL:
   "DB353_M_UNIT_01_STA_4".M_CODES_UNIT_01_STA_4.READ_IN_DISABLE_GENERAL := NOT (NOT "DB353_M_UNIT_01_STA_4".M_CODES_UNIT_01_STA_4.M100 AND NOT "DB353_M_UNIT_01_STA_4".M_CODES_UNIT_01_STA_4.M101 AND NOT "DB353_M_UNIT_01_STA_4".M_CODES_UNIT_01_STA_4.M102 AND NOT "DB353_M_UNIT_01_STA_4".M_CODES_UNIT_01_STA_4.M103 AND NOT "DB353_M_UNIT_01_STA_4".M_CODES_UNIT_01_STA_4.M130 AND NOT "DB353_M_UNIT_01_STA_4".M_CODES_UNIT_01_STA_4.M131 AND NOT "DB353_M_UNIT_01_STA_4".M_CODES_UNIT_01_STA_4.M251);
END_REGION
END_FUNCTION
